	ConsumedTotal:			DINT;				(*$H_R desc := Real time total material consumption for this order; $*)
	ConsumedCart:			DINT;				(*$H_R desc := Real time material consumption from the current cart; $*)
															
END_STRUCT
END_TYPE

// ---- Application/CSP/Customer Interface/csp_customerInterfaces_casePackerCtCall.TcDUT
(*********************************** G.D S.p.A. - Technical Department ***********************************
============= PROGRAM INFO ============
FOLDER:             TBD
MACHINES INVOLVED:  TBD 

============= DESCRIPTION =============
Machine declaration

============= REVISIONS ===============
Date		Version	 	Author      	Description             
----------	-------		------------  	--------------------------------------------
2019/03/27 	0000.00	 	CEC 			Creation of the PRG

**********************************************************************************************************)

TYPE csp_customerInterfaces_casePackerCtCall :
STRUCT
	
	LowCaseSupply:			BOOL;				(*$H_R desc := Connected Technician call - Low Case blank supply; $*)
	LowGlueSupply:			BOOL;				(*$H_R desc := Connected Technician call - Low glue supply; $*)
	LowLabelSupply:			BOOL;				(*$H_R desc := Connected Technician call - Low label supply; $*)
	FullScrapBin:			BOOL;				(*$H_R desc := Connected Technician call - Full machine scrap/waste bin; $*)
	FaultedMain:			BOOL;				(*$H_R desc := Connected Technician call - Main machine is faulted; $*)
	FaultedCaseSupply:		BOOL;				(*$H_R desc := Connected Technician call - Local case blank supply system is faulted; $*)
	TBD1:					BOOL;				(*$H_R desc := Connected Technician call - TBD; $*)
	TBD2:					BOOL;				(*$H_R desc := Connected Technician call - TBD; $*)
	TBD3:					BOOL;				(*$H_R desc := Connected Technician call - TBD; $*)
															
END_STRUCT
END_TYPE

// ---- Application/CSP/Customer Interface/csp_customerInterfaces_casePackerDock.TcDUT
(*********************************** G.D S.p.A. - Technical Department ***********************************
============= PROGRAM INFO ============
FOLDER:             TBD
MACHINES INVOLVED:  TBD 

============= DESCRIPTION =============
Machine declaration

============= REVISIONS ===============
Date		Version	 	Author      	Description             
----------	-------		------------  	--------------------------------------------
2019/03/27 	0000.00	 	CEC 			Creation of the PRG

**********************************************************************************************************)

TYPE csp_customerInterfaces_casePackerDock :
STRUCT
	
	DropAvailable:		BOOL;				(*$H_R desc := Dock [x] is available for cart drop; $*)
	PickAvailable:		BOOL;				(*$H_R desc := Dock [x] is available for cart pick; $*)
	Active:				BOOL;				(*$H_R desc := Dock [x] is actively being consumed; $*)
	EntryReq:			BOOL;				(*$H_RW	act_when := IMMEDIATE ;
														desc := AMR is at Dock [x] and ready to drop or pick; $*)
	EntryAck:			BOOL;				(*$H_R desc := Workcell acknowledge entry request [Future use]; $*)
	EntryOK:			BOOL;				(*$H_R desc := OK for AMR to enter dock; $*)
	AmrExited:			BOOL;				(*$H_RW	act_when := IMMEDIATE ;
														desc := AMR has exited the dock; $*)
															
END_STRUCT
END_TYPE

// ---- Application/CSP/Customer Interface/csp_customerInterfaces_casePackerLabels.TcDUT
(*********************************** G.D S.p.A. - Technical Department ***********************************
============= PROGRAM INFO ============
FOLDER:             TBD
MACHINES INVOLVED:  TBD 

============= DESCRIPTION =============
Machine declaration

============= REVISIONS ===============
Date		Version	 	Author      	Description             
----------	-------		------------  	--------------------------------------------
2019/03/27 	0000.00	 	CEC 			Creation of the PRG

**********************************************************************************************************)

TYPE csp_customerInterfaces_casePackerLabels :
STRUCT
	
	Consumed:						DINT;				(*$H_R desc := Real time total material consumption for this order; $*)
															
END_STRUCT
END_TYPE

// ---- Application/CSP/Customer Interface/csp_customerInterfaces_casePackerProdRej.TcDUT
(*********************************** G.D S.p.A. - Technical Department ***********************************
============= PROGRAM INFO ============
FOLDER:             TBD
MACHINES INVOLVED:  TBD 

============= DESCRIPTION =============
Machine declaration

============= REVISIONS ===============
Date		Version	 	Author      	Description             
----------	-------		------------  	--------------------------------------------
2019/03/27 	0000.00	 	CEC 			Creation of the PRG

**********************************************************************************************************)

TYPE csp_customerInterfaces_casePackerProdRej :
STRUCT
	
	
	Infeed_waterfall:			DINT;				(*$H_R desc := REAL TIME Itemized scrap FOR THIS order; $*)
	Accumulator:				DINT;				(*$H_R desc := REAL TIME Itemized scrap FOR THIS order; $*)
	Case_Feed:					DINT;				(*$H_R desc := REAL TIME Itemized scrap FOR THIS order; $*)
	Discharge:					DINT;				(*$H_R desc := REAL TIME Itemized scrap FOR THIS order; $*)
	TBD5:						DINT;				(*$H_R desc := REAL TIME Itemized scrap FOR THIS order; $*)
	Sample:						DINT;				(*$H_R desc := REAL TIME Itemized scrap FOR THIS order; $*)

															
END_STRUCT
END_TYPE

// ---- Application/CSP/Customer Interface/csp_customerInterfaces_casePackerProduction.TcDUT
(*********************************** G.D S.p.A. - Technical Department ***********************************
============= PROGRAM INFO ============
FOLDER:             TBD
MACHINES INVOLVED:  TBD 

============= DESCRIPTION =============
Machine declaration

============= REVISIONS ===============
Date		Version	 	Author      	Description             
----------	-------		------------  	--------------------------------------------
2019/03/27 	0000.00	 	CEC 			Creation of the PRG

**********************************************************************************************************)

TYPE csp_customerInterfaces_casePackerProduction :
STRUCT
	
	TotalUnits:			DINT;									(*$H_R desc := Real time total number of cartons received for this order; $*)
	GoodPods:			DINT;									(*$H_R desc := Real time total number of good pods packed for this order; $*)
	GoodUnits:			DINT;									(*$H_R desc := Real time total number of good cartons made for this order; $*)
	GoodCases:			DINT;									(*$H_R desc := Real time total number of good cases made for this order; $*)
	TotalUnitsNoReset:	DINT;									(*$H_R desc := Real time total number of cartons received, reset to 1 after 4294967295; $*)
	GoodPodsNoReset:	DINT;									(*$H_R desc := Real time total number of good pods, reset to 1 after 4294967295; $*)
	GoodUnitsNoReset:	DINT;									(*$H_R desc := Real time total number of good cartons, reset to 1 after 4294967295; $*)
	GoodCasesNoReset:	DINT;									(*$H_R desc := Real time total number of good cases, reset to 1 after 4294967295; $*)
	TotalScrapUnits:	DINT;									(*$H_R desc := Real time total number of scrap cartons rejected; $*)
	TotalOrderTime:		DINT;									(*$H_R desc := Real time total minute counter for current order; $*)
	TotalRunningTime:	DINT;									(*$H_R desc := Real time total minute counter for running time in current order; $*)
	PercentScrapUnits:	DINT;									(*$H_R desc := Real time percentage of total cartons rejected; $*)
	Rejects:			csp_customerInterfaces_casePackerProdRej;
															
END_STRUCT
END_TYPE

// ---- Application/CSP/Customer Interface/csp_customerInterfaces_casePackerStart.TcDUT
(*********************************** G.D S.p.A. - Technical Department ***********************************
============= PROGRAM INFO ============
FOLDER:             TBD
MACHINES INVOLVED:  TBD 

============= DESCRIPTION =============
Machine declaration

============= REVISIONS ===============
Date		Version	 	Author      	Description             
----------	-------		------------  	--------------------------------------------
2019/03/27 	0000.00	 	CEC 			Creation of the PRG

**********************************************************************************************************)

TYPE csp_customerInterfaces_casePackerStart :
STRUCT
	
	Request:					BOOL;				(*$H_R desc := Machine request FOR permission TO start; $*)
	Ramp:						BOOL;				(*$H_R desc := Machine is in high current start-up ramp; $*)
	PeakWait:					BOOL;				(*$H_RW	act_when := IMMEDIATE ;
															desc := Request FROM SCADA FOR machine TO delay start; $*)
															
END_STRUCT
END_TYPE

// ---- Application/CSP/Customer Interface/csp_customerInterfaces_casePackerStatus.TcDUT
(*********************************** G.D S.p.A. - Technical Department ***********************************
============= PROGRAM INFO ============
FOLDER:             TBD
MACHINES INVOLVED:  TBD 

============= DESCRIPTION =============
Machine declaration

============= REVISIONS ===============
Date		Version	 	Author      	Description             
----------	-------		------------  	--------------------------------------------
2019/03/27 	0000.00	 	CEC 			Creation of the PRG

**********************************************************************************************************)

TYPE csp_customerInterfaces_casePackerStatus :
STRUCT
	
	Online:					BOOL;				(*$H_R desc := Machine is online; $*)
	Job:					DINT;				(*$H_R desc := Current order (Job) status; $*)
	NextJob:				DINT;				(*$H_R desc := Next order (Job) status; $*)
	Running:				BOOL;				(*$H_R desc := Machine is actively making product; $*)
	Faulted:				csp_customerInterfaces_casePackerStFault;
	RunOut:					BOOL;				(*$H_R desc := Machine AND  conveyor clearance in process; $*)
	RunOutComplete:			BOOL;				(*$H_R desc := Machine AND conveyor clearance complete; $*)
	Rate:					csp_customerInterfaces_casePackerStRate;
	Stop:					csp_customerInterfaces_casePackerStStop;
	Starved:				csp_customerInterfaces_casePackerStStarved;
	Blocked:				csp_customerInterfaces_casePackerStBlocked;
															
END_STRUCT
END_TYPE

// ---- Application/CSP/Customer Interface/csp_customerInterfaces_casePackerStBlocked.TcDUT
(*********************************** G.D S.p.A. - Technical Department ***********************************
============= PROGRAM INFO ============
FOLDER:             TBD
MACHINES INVOLVED:  TBD 

============= DESCRIPTION =============
Machine declaration

============= REVISIONS ===============
Date		Version	 	Author      	Description             
----------	-------		------------  	--------------------------------------------
2019/03/27 	0000.00	 	CEC 			Creation of the PRG

**********************************************************************************************************)

TYPE csp_customerInterfaces_casePackerStBlocked :
STRUCT
	
	Downstream:	BOOL;				(*$H_R desc := Stopped due TO downstream backup; $*)
	Reject:		BOOL;				(*$H_R desc := Stopped due TO scrap backup; $*)
	Waste:		BOOL;				(*$H_R desc := Stopped due TO waste backup; $*)
															
END_STRUCT
END_TYPE

// ---- Application/CSP/Customer Interface/csp_customerInterfaces_casePackerStFault.TcDUT
(*********************************** G.D S.p.A. - Technical Department ***********************************
============= PROGRAM INFO ============
FOLDER:             TBD
MACHINES INVOLVED:  TBD 

============= DESCRIPTION =============
Machine declaration

============= REVISIONS ===============
Date		Version	 	Author      	Description             
----------	-------		------------  	--------------------------------------------
2019/03/27 	0000.00	 	CEC 			Creation of the PRG

**********************************************************************************************************)

TYPE csp_customerInterfaces_casePackerStFault :
STRUCT
	
	Main:				BOOL;				(*$H_R desc := Main machine is faulted; $*)
	CaseBlanks:			BOOL;				(*$H_R desc := Local case blank supply system is faulted; $*)
															
END_STRUCT
END_TYPE

// ---- Application/CSP/Customer Interface/csp_customerInterfaces_casePackerStRate.TcDUT
(*********************************** G.D S.p.A. - Technical Department ***********************************
============= PROGRAM INFO ============
FOLDER:             TBD
MACHINES INVOLVED:  TBD 

============= DESCRIPTION =============
Machine declaration

============= REVISIONS ===============
Date		Version	 	Author      	Description             
----------	-------		------------  	--------------------------------------------
2019/03/27 	0000.00	 	CEC 			Creation of the PRG

**********************************************************************************************************)

TYPE csp_customerInterfaces_casePackerStRate :
STRUCT
	
	Target:			INT;				(*$H_R desc := Target rate in Pods/minute; $*)
	Actual:			INT;				(*$H_R desc := REAL-TIME rate in Pods/minute; $*)
															
END_STRUCT
END_TYPE

// ---- Application/CSP/Customer Interface/csp_customerInterfaces_casePackerStStarved.TcDUT
(*********************************** G.D S.p.A. - Technical Department ***********************************
============= PROGRAM INFO ============
FOLDER:             TBD
MACHINES INVOLVED:  TBD 

============= DESCRIPTION =============
Machine declaration

============= REVISIONS ===============
Date		Version	 	Author      	Description             
----------	-------		------------  	--------------------------------------------
2019/03/27 	0000.00	 	CEC 			Creation of the PRG

**********************************************************************************************************)

TYPE csp_customerInterfaces_casePackerStStarved :
STRUCT
	
	Units:			BOOL;				(*$H_R desc := Carton infeed is empty due to upstream supply; $*)
	CaseBlanks:		BOOL;				(*$H_R desc := Case blank infeed is empty due to upstream supply; $*)
	Glue:			BOOL;				(*$H_R desc := Glue hopper is empty; $*)
	Labels:			BOOL;				(*$H_R desc := Case labeler reel is empty; $*)
															
END_STRUCT
END_TYPE

// ---- Application/CSP/Customer Interface/csp_customerInterfaces_casePackerStStop.TcDUT
(*********************************** G.D S.p.A. - Technical Department ***********************************
============= PROGRAM INFO ============
FOLDER:             TBD
MACHINES INVOLVED:  TBD 

============= DESCRIPTION =============
Machine declaration

============= REVISIONS ===============
Date		Version	 	Author      	Description             
----------	-------		------------  	--------------------------------------------
2019/03/27 	0000.00	 	CEC 			Creation of the PRG

**********************************************************************************************************)

TYPE csp_customerInterfaces_casePackerStStop :
STRUCT
	
	AutoReason:		DINT;				(*$H_R desc := Automatically collected reason FOR current downtime; $*)
	Estop:			BOOL;				(*$H_R desc := Current downtime a result OF Estop; $*)
	Guard:			BOOL;				(*$H_R desc := Current downtime a result OF guard trip; $*)
	Operator:		BOOL;				(*$H_R desc := Current downtime a result OF normal operator stop; $*)
															
END_STRUCT
END_TYPE

// ---- Application/CSP/Customer Interface/csp_customerInterfaces_fillWeight.TcDUT
(*********************************** G.D S.p.A. - Technical Department ***********************************
============= PROGRAM INFO ============
FOLDER:             TBD
MACHINES INVOLVED:  TBD 

============= DESCRIPTION =============
Machine declaration

============= REVISIONS ===============
Date		Version	 	Author      	Description             
----------	-------		------------  	--------------------------------------------
2019/03/27 	0000.00	 	CEC 			Creation of the PRG

**********************************************************************************************************)

TYPE csp_customerInterfaces_fillWeight :
STRUCT
	
	Target:				REAL;				(*$H_RW	act_when := IMMEDIATE ;
															desc := Ingredient fill weight; $*)
	Maximum:			REAL;				(*$H_RW	act_when := IMMEDIATE ;
															desc := Ingredient max weight; $*)
	Minimum:			REAL;				(*$H_RW	act_when := IMMEDIATE ;
															desc := Ingredient min weight; $*)
	
END_STRUCT
END_TYPE

// ---- Application/CSP/Customer Interface/csp_customerInterfaces_mark.TcDUT
(*********************************** G.D S.p.A. - Technical Department ***********************************
============= PROGRAM INFO ============
FOLDER:             TBD
MACHINES INVOLVED:  TBD 

============= DESCRIPTION =============
Machine declaration

============= REVISIONS ===============
Date		Version	 	Author      	Description             
----------	-------		------------  	--------------------------------------------
2019/03/27 	0000.00	 	CEC 			Creation of the PRG

**********************************************************************************************************)

TYPE csp_customerInterfaces_mark :
STRUCT
	
	ID:								STRING;				(*$H_RW	act_when := IMMEDIATE ;
															desc := Print job ID FROM MES; $*)
	BUBD:							csp_customerInterfaces_markBUBD;
		
	OriginDate:						STRING;				(*$H_RW	act_when := IMMEDIATE ;
															desc := DATE the Pod was manufactured; $*)					
	DestCode:						STRING;				(*$H_RW	act_when := IMMEDIATE ;
															desc := Localization code FOR destination; $*)					
	PartnerSite:					STRING;				(*$H_RW	act_when := IMMEDIATE ;
															desc := Partner site code; $*)	
	KdpSite: 						STRING; 			(*$H_RW act_when := IMMEDIATE ;
															desc := KDP site code; $*)				
	Template:						csp_customerInterfaces_markTemplate;
															
															
END_STRUCT
END_TYPE

// ---- Application/CSP/Customer Interface/csp_customerInterfaces_markBUBD.TcDUT
(*********************************** G.D S.p.A. - Technical Department ***********************************
============= PROGRAM INFO ============
FOLDER:             TBD
MACHINES INVOLVED:  TBD 

============= DESCRIPTION =============
Machine declaration

============= REVISIONS ===============
Date		Version	 	Author      	Description             
----------	-------		------------  	--------------------------------------------
2019/03/27 	0000.00	 	CEC 			Creation of the PRG

**********************************************************************************************************)

TYPE csp_customerInterfaces_markBUBD :
STRUCT
	
	BestUsedByDate:			STRING;				(*$H_RW	act_when := IMMEDIATE ;
															desc := Best Used BY DATE; $*)													
	BestUsedByDate_Short:	STRING;				(*$H_RW	act_when := IMMEDIATE ;
															desc := Best Used BY DATE; $*)													
	Prefix:					STRING;				(*$H_RW	act_when := IMMEDIATE ;
															desc := BUBD Prefix (abbreviation); $*)	
	Format:					STRING;				(*$H_RW	act_when := IMMEDIATE ;
															desc := BUBD localized DATE format; $*)		
															
END_STRUCT
END_TYPE

// ---- Application/CSP/Customer Interface/csp_customerInterfaces_markTemplate.TcDUT
(*********************************** G.D S.p.A. - Technical Department ***********************************
============= PROGRAM INFO ============
FOLDER:             TBD
MACHINES INVOLVED:  TBD 

============= DESCRIPTION =============
Machine declaration

============= REVISIONS ===============
Date		Version	 	Author      	Description             
----------	-------		------------  	--------------------------------------------
2019/03/27 	0000.00	 	CEC 			Creation of the PRG

**********************************************************************************************************)

TYPE csp_customerInterfaces_markTemplate :
STRUCT
	
	Pod:					STRING;				(*$H_RW	act_when := IMMEDIATE ;
														desc := Filler product mark template [future use]; $*)				
	Carton:					STRING;				(*$H_RW	act_when := IMMEDIATE ;
														desc := Cartoner product mark template [future use]; $*)					
	CASEPACK:				STRING;				(*$H_RW	act_when := IMMEDIATE ;
														desc := CASE packer product mark template [future use]; $*)	
							
															
END_STRUCT
END_TYPE

// ---- Application/CSP/Customer Interface/csp_customerInterfaces_material.TcDUT
(*********************************** G.D S.p.A. - Technical Department ***********************************
============= PROGRAM INFO ============
FOLDER:             TBD
MACHINES INVOLVED:  TBD 

============= DESCRIPTION =============
Machine declaration

============= REVISIONS ===============
Date		Version	 	Author      	Description             
----------	-------		------------  	--------------------------------------------
2019/03/27 	0000.00	 	CEC 			Creation of the PRG

**********************************************************************************************************)

TYPE csp_customerInterfaces_material :
STRUCT
	
	ID:							STRING;				(*$H_RW	act_when := IMMEDIATE ;
															desc := Material ID in current order; $*)
	QTY:						REAL;				(*$H_RW	act_when := IMMEDIATE ;
															desc := Total expected material QTY for current order; $*)
															
END_STRUCT
END_TYPE

// ---- Application/CSP/Customer Interface/csp_customerInterfaces_MES.TcDUT
(*********************************** G.D S.p.A. - Technical Department ***********************************
============= PROGRAM INFO ============
FOLDER:             TBD
MACHINES INVOLVED:  TBD 

============= DESCRIPTION =============
Machine declaration

============= REVISIONS ===============
Date		Version	 	Author      	Description             
----------	-------		------------  	--------------------------------------------
2019/03/27 	0000.00	 	CEC 			Creation of the PRG

**********************************************************************************************************)

TYPE csp_customerInterfaces_MES :
STRUCT

	StartJobReq:					BOOL;				(*$H_RW	act_when := IMMEDIATE ;
															desc := Request FROM MES TO start the current job; $*)				
	RunOutReq:						BOOL;				(*$H_RW	act_when := IMMEDIATE ;
															desc := Request FROM MES TO execute a line clearance; $*)				
	EndJobReq:						BOOL;				(*$H_RW	act_when := IMMEDIATE ;
															desc := Request FROM MES TO end the current job; $*)					
	CycleEnable:					BOOL;				(*$H_RW	act_when := IMMEDIATE ;
															desc := Premissive FROM MES TO run the line; $*)					
	Alarm:							DINT;				(*$H_RW	act_when := IMMEDIATE ;
															desc := Predefined alarms FROM MES; $*)					
	Warning:						DINT;				(*$H_RW	act_when := IMMEDIATE ;
															desc := Predefined warnings/messages FROM MES; $*)				
															
END_STRUCT
END_TYPE

// ---- Application/CSP/Customer Interface/csp_customerInterfaces_order.TcDUT
(*********************************** G.D S.p.A. - Technical Department ***********************************
============= PROGRAM INFO ============
FOLDER:             TBD
MACHINES INVOLVED:  TBD 

============= DESCRIPTION =============
Machine declaration

============= REVISIONS ===============
Date		Version	 	Author      	Description             
----------	-------		------------  	--------------------------------------------
2019/03/27 	0000.00	 	CEC 			Creation of the PRG

**********************************************************************************************************)

TYPE csp_customerInterfaces_order :
STRUCT
	
	ID:								STRING;				(*$H_RW	act_when := IMMEDIATE ;
															desc := product order identifier; $*)
	SapBatchID:						STRING;				(*$H_RW	act_when := IMMEDIATE ;
															desc := SAP batch ID; $*)
	
END_STRUCT
END_TYPE

// ---- Application/CSP/Customer Interface/csp_customerInterfaces_palletizer.TcDUT
(*********************************** G.D S.p.A. - Technical Department ***********************************
============= PROGRAM INFO ============
FOLDER:             TBD
MACHINES INVOLVED:  TBD 

============= DESCRIPTION =============
Machine declaration

============= REVISIONS ===============
Date		Version	 	Author      	Description             
----------	-------		------------  	--------------------------------------------
2019/03/27 	0000.00	 	CEC 			Creation of the PRG

**********************************************************************************************************)

TYPE csp_customerInterfaces_palletizer :
STRUCT
	
	Ready:				BOOL;			(*$H_RW	act_when := IMMEDIATE ;
															desc := Palletizer is ready to receive cases; $*)
															
END_STRUCT
END_TYPE

// ---- Application/CSP/Customer Interface/csp_customerInterfaces_product.TcDUT
(*********************************** G.D S.p.A. - Technical Department ***********************************
============= PROGRAM INFO ============
FOLDER:             TBD
MACHINES INVOLVED:  TBD 

============= DESCRIPTION =============
Machine declaration

============= REVISIONS ===============
Date		Version	 	Author      	Description             
----------	-------		------------  	--------------------------------------------
2019/03/27 	0000.00	 	CEC 			Creation of the PRG

**********************************************************************************************************)

TYPE csp_customerInterfaces_product :
STRUCT
	
	ID:							STRING;				(*$H_RW	act_when := IMMEDIATE ;
														desc := Product ID; $*)
	UPC:						STRING;				(*$H_RW	act_when := IMMEDIATE ;
														desc := Product UPC; $*)
	
	PodsPerCarton: 				INT;				(*$H_RW	act_when := IMMEDIATE ;
															desc := recipe data, number of cups inside a carton; $*)
	
	PodsPerCase:				INT;				(*$H_RW	act_when := IMMEDIATE ;
															desc := recipe data, number of cups inside a case; $*)
	CartonsPerCase:				INT;				(*$H_RW	act_when := IMMEDIATE ;
															desc := recipe data, number of cartons inside a case; $*)

	FillWeight:					csp_customerInterfaces_fillWeight;

	FilterType:					STRING;				(*$H_RW	act_when := IMMEDIATE ;
															desc := Filter type; $*)
	CaffeinatedFlag:			BOOL;				(*$H_RW	act_when := IMMEDIATE ;
															desc := Coffee Caffeinated flag; $*)
	KosherFlag:					BOOL;				(*$H_RW	act_when := IMMEDIATE ;
															desc := Coffee Kosher flag; $*)
	OrganicFlag:				BOOL;				(*$H_RW	act_when := IMMEDIATE ;
															desc := Coffee Organic flag; $*)
	FlavorFlag:					BOOL;				(*$H_RW	act_when := IMMEDIATE ;
															desc := Coffee Flavored flag; $*)
	FlavorDose:					REAL;				(*$H_RW	act_when := IMMEDIATE ;
															desc := Coffee inline flavor dose [future use]; $*)
	ShelfLife:					INT;				(*$H_RW	act_when := IMMEDIATE ;
															desc := Pod shelf life; $*)
	
END_STRUCT
END_TYPE

// ---- Application/CSP/Customer Interface/csp_customerInterfaces_recipe.TcDUT
(*********************************** G.D S.p.A. - Technical Department ***********************************
============= PROGRAM INFO ============
FOLDER:             TBD
MACHINES INVOLVED:  TBD 

============= DESCRIPTION =============
Machine declaration

============= REVISIONS ===============
Date		Version	 	Author      	Description             
----------	-------		------------  	--------------------------------------------
2019/03/27 	0000.00	 	CEC 			Creation of the PRG

**********************************************************************************************************)

TYPE csp_customerInterfaces_recipe :
STRUCT
	
	Filler:								STRING;				(*$H_RW	act_when := IMMEDIATE ;
															desc := Filler recipe ID [future use]; $*)
	Cartoner:							STRING;				(*$H_RW	act_when := IMMEDIATE ;
															desc := Cartoner recipe ID [future use]; $*)
	CasePacker:							STRING;				(*$H_RW	act_when := IMMEDIATE ;
															desc := Case packer recipe ID [future use]; $*)
															
END_STRUCT
END_TYPE

// ---- Application/CSP/Main/AccU Change/csp_main_accuChange_constant.TcDUT
TYPE csp_main_accuChange_constant :
STRUCT
	(*BELT Info*)
	MIN_VELOCITY_MMpSEC:						LREAL := 100;
	MAX_VELOCITY_MMpSEC:						LREAL := 666.5487;
	MAX_ACCELERATION_MMpSEC2:					LREAL := 1000;
	MAX_DECELERATION_MMpSEC2:					LREAL := 1000;
	MAX_JERK_MMpSEC3:							LREAL := 100000;
	RUNNING_ACCELERATION_MMMpSEC2:				LREAL := 3000;
	RUNNING_DECELERATION_MMpSEC2:				LREAL := 3000;
	MAX_FOLLOWING_ERROR_MM:						LREAL := 5;
	
	RUNNING_JERK_MMpSEC3:						LREAL := 1000000;
	MOTOR_MAX_VELOCITY_DEGPS:					LREAL := 9600;
	MOTOR_MAX_ACCELERATION_DEGPS2:				LREAL := 4800;
	MOTOR_MAX_DECELERATION_DEGPS2:				LREAL := 4800;
	MOTOR_MAX_JERK_DEGPS3:						LREAL := 100000000; 
	MOTOR_MAX_FOLLOWING_ERROR_DEG:				LREAL := 2;
END_STRUCT
END_TYPE

// ---- Application/CSP/Main/AccU Change/csp_main_accuChange_enum.TcDUT
TYPE csp_main_accuChange_enum :
(
	CSP_MAIN_ACCUCHANGE_STATUS_BRAND_CHECK 									:= 0,
	CSP_MAIN_ACCUCHANGE_STATUS_BRAND_CHANGE_REQUEST 						:= 5,
	CSP_MAIN_ACCUCHANGE_STATUS_PRODUCT_REMOVED_CHECK 						:= 10,
	CSP_MAIN_ACCUCHANGE_STATUS_RESET_REQUEST								:= 20,
	CSP_MAIN_ACCUCHANGE_STATUS_SAFE_POSITION_REQUEST 						:= 30,
	CSP_MAIN_ACCUCHANGE_STATUS_OPERATOR_REPLACE_CHANGE_PARTS 				:= 40,
	CSP_MAIN_ACCUCHANGE_STATUS_CHANGE_PARTS_REPLACED						:= 50,
	CSP_MAIN_ACCUCHANGE_STATUS_VERIFYING_CHANGE_PARTS_START					:= 60,
	CSP_MAIN_ACCUCHANGE_STATUS_VERIFYING_CASE_FEED_EOAT						:= 61,
	CSP_MAIN_ACCUCHANGE_STATUS_VERIFYING_LOADER_PUSHER						:= 62,
	CSP_MAIN_ACCUCHANGE_STATUS_VERIFYING_LOADER_GUIDE_PLATE					:= 63,
	CSP_MAIN_ACCUCHANGE_STATUS_VERIFYING_CLOSING_PADDLES					:= 64,
	CSP_MAIN_ACCUCHANGE_STATUS_VERIFYING_ALL_RFID							:= 65,
	CSP_MAIN_ACCUCHANGE_STATUS_GROUP_1_ACCU_MOVE_REQUEST 					:= 70,
	CSP_MAIN_ACCUCHANGE_STATUS_GROUP_2_TR_UP_ACCU_MOVE_REQUEST 				:= 80,
	CSP_MAIN_ACCUCHANGE_STATUS_GROUP_2_TR_DOWN_ACCU_MOVE_REQUEST 			:= 85,
	CSP_MAIN_ACCUCHANGE_STATUS_ADD_CASE_BLANKS 								:= 100,
	CSP_MAIN_ACCUCHANGE_STATUS_DONE											:= 900
) := CSP_MAIN_ACCUCHANGE_STATUS_BRAND_CHECK;
END_TYPE

// ---- Application/CSP/Main/AccU Change/csp_main_accuChange_partColor_enum.TcDUT
TYPE csp_main_accuChange_partColor_enum :
(
	NO_COLOR		 	:= 0,
	RED					:= 1,
	GREEN				:= 2,
	BLUE				:= 3,
	YELLOW				:= 4,
	WHITE				:= 5,
	BLACK				:= 6,
	ORANGE				:= 7
);
END_TYPE

// ---- Application/CSP/Main/AccU Change/csp_main_accuChange_RFID_reader_list.TcDUT
TYPE csp_main_accuChange_RFID_reader_list :
(
	NO_READER_SELECTED							:= 0,
	CASE_FEED_EOAT_READER						:= 1,
	LOADER_PUSHER_READER						:= 2, (* IN CODE *)
	LOADER_GUIDE_PLATE_READER					:= 3, (* IN CODE *)
	CLOSING_PADDLES_READER						:= 4  (* IN CODE *)
):= NO_READER_SELECTED;
END_TYPE

// ---- Application/CSP/Main/AccU Change/csp_main_accuChange_RFID_read_write_status.TcDUT
TYPE csp_main_accuChange_RFID_read_write_status :
(
	READ_WRITE_STATUS_START_RFID_READ						:= 0,
	READ_WRITE_STATUS_SEND_READ_COMMAND						:= 1,
	READ_WRITE_STATUS_WAIT_FOR_READ_RESULT					:= 2,
	READ_WRITE_STATUS_CHECK_READ_RESULT						:= 3,
	
	READ_WRITE_STATUS_START_RFID_WRITE						:= 101,
	READ_WRITE_STATUS_SEND_WRITE_COMMAND					:= 102,
	READ_WRITE_STATUS_WAIT_FOR_WRITE_SUCCESS				:= 103,
	READ_WRITE_STATUS_WRITE_TO_READ							:= 104,
	
	READ_WRITE_STATUS_WAITING								:= 900,
	READ_WRITE_STATUS_ERROR									:= 999
):= READ_WRITE_STATUS_WAITING;
END_TYPE

// ---- Application/CSP/Main/AccU Change/csp_main_accuChange_RFID_running_check_status.TcDUT
TYPE csp_main_accuChange_RFID_running_check_status :
(
	READ_RUNNING_CHECK_STATUS_START									:= 0,
	READ_RUNNING_CHECK_STATUS_EOAT_CHECK_CP							:= 1,
	READ_RUNNING_CHECK_STATUS_EOAT_SEND_READ						:= 2,
	READ_RUNNING_CHECK_STATUS_EOAT_CHECK_READ						:= 3,
	READ_RUNNING_CHECK_STATUS_LOADER_PUSHER_CHECK_CP				:= 4,
	READ_RUNNING_CHECK_STATUS_LOADER_PUSHER_SEND_READ				:= 5,
	READ_RUNNING_CHECK_STATUS_LOADER_PUSHER_CHECK_READ				:= 6,
	READ_RUNNING_CHECK_STATUS_LOADER_PLATE_CHECK_CP					:= 7,
	READ_RUNNING_CHECK_STATUS_LOADER_PLATE_SEND_READ				:= 8,
	READ_RUNNING_CHECK_STATUS_LOADER_PLATE_CHECK_READ				:= 9,
	
	READ_RUNNING_CHECK_STATUS_DONE									:= 900,
	READ_RUNNING_CHECK_STATUS_WAITING								:= 950,
	READ_RUNNING_CHECK_STATUS_ERROR									:= 999
):= READ_RUNNING_CHECK_STATUS_WAITING;
END_TYPE

// ---- Application/CSP/Main/Brand/csp_main_brand_cam_change.TcDUT
TYPE csp_main_brand_cam_change :
(
	CSP_MAIN_BRAND_CAM_CHANGE_INIT 							:= 0,
	CSP_MAIN_BRAND_CAM_CHANGE_PHASE_LOAD 					:= 10,
	CSP_MAIN_BRAND_CAM_CHANGE_PHASE_TRANSFER 				:= 20,
	CSP_MAIN_BRAND_CAM_CHANGE_CONNEECTION_LOAD 				:= 30,
	CSP_MAIN_BRAND_CAM_CHANGE_CONNECTION_TRANSFER 			:= 40,		
	CSP_MAIN_BRAND_CAM_CHANGE_DONE							:= 900,
	CSP_MAIN_BRAND_CAM_CHANGE_ERROR							:= 999
) := CSP_MAIN_BRAND_CAM_CHANGE_INIT;
END_TYPE

// ---- Application/CSP/Main/Brand/csp_main_brand_carton_format_enum.TcDUT
TYPE csp_main_brand_carton_format_enum :
	(
		csp_MAIN_BRAND_X_COUNT_XxXCARTON_X_COUNT_CASE  	:= 0,
		csp_MAIN_BRAND_6_COUNT_2x3CARTON_6_COUNT_CASE  	:= 1,
		csp_MAIN_BRAND_8_COUNT_2x4CARTON_6_COUNT_CASE  	:= 2,
		csp_MAIN_BRAND_10_COUNT_2x3CARTON_6_COUNT_CASE	:= 3,
		csp_MAIN_BRAND_12_COUNT_2x3CARTON_6_COUNT_CASE	:= 4,
		csp_MAIN_BRAND_16_COUNT_2x3CARTON_4_COUNT_CASE	:= 5,
		csp_MAIN_BRAND_18_COUNT_2x3CARTON_4_COUNT_CASE	:= 6,
		csp_MAIN_BRAND_14_COUNT_2x4CARTON_6_COUNT_CASE	:= 7,
		csp_MAIN_BRAND_16_COUNT_2x4CARTON_6_COUNT_CASE	:= 8,
		csp_MAIN_BRAND_20_COUNT_2x4CARTON_4_COUNT_CASE	:= 9,
		csp_MAIN_BRAND_22_COUNT_2x4CARTON_4_COUNT_CASE	:= 10,
		csp_MAIN_BRAND_24_COUNT_2x4CARTON_4_COUNT_CASE	:= 11,
		csp_MAIN_BRAND_28_COUNT_2x4CARTON_4_COUNT_CASE	:= 12,
		csp_MAIN_BRAND_30_COUNT_2x4CARTON_4_COUNT_CASE	:= 13,
		csp_MAIN_BRAND_32_COUNT_2x4CARTON_4_COUNT_CASE	:= 14,
		csp_MAIN_BRAND_34_COUNT_3x4CARTON_4_COUNT_CASE	:= 15,
		csp_MAIN_BRAND_36_COUNT_3x4CARTON_4_COUNT_CASE	:= 16,		
		csp_MAIN_BRAND_44_COUNT_3x4CARTON_4_COUNT_CASE	:= 17,
		csp_MAIN_BRAND_46_COUNT_3x4CARTON_4_COUNT_CASE	:= 18,
		csp_MAIN_BRAND_48_COUNT_3x4CARTON_4_COUNT_CASE	:= 19
	
	) := csp_MAIN_BRAND_X_COUNT_XxXCARTON_X_COUNT_CASE;
END_TYPE

// ---- Application/CSP/Main/Brand/csp_main_brand_case_pattern.TcDUT
TYPE csp_main_brand_case_pattern :
STRUCT
	
	case_pattern_L:								INT := 2; (*$P min := 0; max := 5; step := 1; unit := u ; desc := Case Pattern L; $*)
	case_pattern_W:								INT := 2; (*$P min := 0; max := 5; step := 1; unit := u; desc := Case Pattern W; $*)
	case_pattern_D:								INT := 1; (*$P min := 0; max := 5; step := 1; unit := u; desc := Case Pattern D; $*)
			
END_STRUCT
END_TYPE

// ---- Application/CSP/Main/Brand/csp_main_brand_product_dimension.TcDUT
TYPE csp_main_brand_product_dimension :
	STRUCT
		
		carton_size_L_mm:								LREAL := 100; (*$P min := 0; max := 200; step := 0.1; unit :=  mm; desc := Carton Length; $*)
		carton_size_W_mm:								LREAL := 100; (*$P min := 0; max := 200; step := 0.1; unit :=  mm; desc := Carton Width; $*)
		carton_size_D_mm:								LREAL := 100; (*$P min := 0; max := 200; step := 0.1; unit :=  mm; desc := Carton Depth; $*)
				
	END_STRUCT
END_TYPE

// ---- Application/CSP/Main/Interface/csp_main_interface_csv_read.TcDUT
{attribute 'qualified_only'}
{attribute 'strict'}
TYPE csp_main_interface_csv_read :
(
	
	csv_read_idle					:= 0,
	csv_read_wait_for_alarm			:= 10,
	csv_read_clear_variables		:= 20,
	csv_read_trim_object_name		:= 30,
	csv_read_open_csv_file			:= 40,
	csv_read_verify_open			:= 50,
	csv_read_read_csv_file			:= 60,
	csv_read_verify_read			:= 70,
	csv_read_parse_csv_stop_data	:= 80,
	csv_read_compare_stop			:= 90,
	csv_read_alarm_found			:= 100,
	csv_read_close_csv_file			:= 200,
	csv_read_close_csv_file_verify	:= 210
	
) := csv_read_idle;
END_TYPE

// ---- Application/CSP/Main/Jog Manager/csp_jog_accu_suggested_speeds.TcDUT
TYPE csp_jog_accu_suggested_speeds :
	STRUCT
		NO_UAXIS_SELECT_TO_JOG_SPEED:															LREAL := 0;
		SMTR61700_TRANSFER_INFEED_DEPTH_SPEED:													LREAL := 1.5;
		SMTR61710_TRANSFER_INFEED_WATERFALL_ADJUST_SPEED:										LREAL := 1;
		SMTR61720_SMTR61730_TRANSFER_ACCUMULATOR_DEPTH_AND_CONVEYOR_DEPTH_SPEED:				LREAL := 1;
		SMTR61510_CASE_TOP_RAIL_DEPTH_SPEED:													LREAL := 2;
		SMTR61430_SMTR61500_CASE_TOP_RAIL_LS_AND_OS_WIDTH_SPEED:								LREAL := 1;
		SMTR61210_SMTR61200_SMTR61420_CASE_FEED_SHUTTLE_TRANSPORT_AND_DISCHARGE_DEPTH_SPEED:	LREAL := 2;
		SMTR61220_CASE_FEED_MAGAZINE_LS_DEPTH_SPEED:											LREAL := 1;
		SMTR61230_CASE_FEED_MAGAZINE_OS_DEPTH_SPEED:											LREAL := 1;
		SMTR61300_CASE_LOADER_GUIDE_WIDTH_SPEED:												LREAL := 5;
		SMTR61410_CASE_GLUE_LS_LOWER_POSITION_SPEED:											LREAL := 3;
		SMTR61400_CASE_GLUE_LS_UPPER_POSITION_SPEED:											LREAL := 3;
		SMTR61330_CASE_GLUE_OS_LOWER_POSITION_SPEED:											LREAL := 3;
		SMTR61320_CASE_GLUE_OS_UPPER_POSITION_SPEED:											LREAL := 3;
		SMTR61310_CASE_GLUE_OS_WIDTH_SPEED:														LREAL := 3;
		
		(*Tie AccuChange axis list enum to each axis' suggested speed
		If accuchange jog list enum is changed, indices here must be adjusted accordingly*)
		Suggested_Speeds:	ARRAY[JOG_MANAGER_JOG_LIST_NONE..JOG_MANAGER_JOG_LIST_MAX] OF LREAL :=
			[NO_UAXIS_SELECT_TO_JOG_SPEED, //0
			SMTR61700_TRANSFER_INFEED_DEPTH_SPEED, //1
			SMTR61710_TRANSFER_INFEED_WATERFALL_ADJUST_SPEED, //2
			SMTR61720_SMTR61730_TRANSFER_ACCUMULATOR_DEPTH_AND_CONVEYOR_DEPTH_SPEED, //3
			0, //4 - csp_jog_list_AccUChange enum has no 4 value
			SMTR61510_CASE_TOP_RAIL_DEPTH_SPEED, //5
			SMTR61430_SMTR61500_CASE_TOP_RAIL_LS_AND_OS_WIDTH_SPEED, //6
			SMTR61210_SMTR61200_SMTR61420_CASE_FEED_SHUTTLE_TRANSPORT_AND_DISCHARGE_DEPTH_SPEED, //7
			SMTR61220_CASE_FEED_MAGAZINE_LS_DEPTH_SPEED, //8
			SMTR61230_CASE_FEED_MAGAZINE_OS_DEPTH_SPEED, //9
			SMTR61300_CASE_LOADER_GUIDE_WIDTH_SPEED, //10
			SMTR61410_CASE_GLUE_LS_LOWER_POSITION_SPEED, //11
			SMTR61400_CASE_GLUE_LS_UPPER_POSITION_SPEED, //12
			SMTR61330_CASE_GLUE_OS_LOWER_POSITION_SPEED, //13
			SMTR61320_CASE_GLUE_OS_UPPER_POSITION_SPEED, //14
			SMTR61310_CASE_GLUE_OS_WIDTH_SPEED]; //15
	
	END_STRUCT
END_TYPE

// ---- Application/CSP/Main/Jog Manager/csp_jog_list_AccUChange.TcDUT
TYPE csp_jog_list_AccUChange :
(	
	JOG_LIST_NO_UAXIS_SELECT_TO_JOG													:= 0,
	SMTR61700_TRANSFER_INFEED_DEPTH													:= 1,
	SMTR61710_TRANSFER_INFEED_WATERFALL_ADJUST										:= 2,
	SMTR61720_SMTR61730_TRANSFER_ACCUMULATOR_DEPTH_AND_CONVEYOR_DEPTH 				:= 3,
	SMTR61510_CASE_TOP_RAIL_DEPTH													:= 5,
	SMTR61430_SMTR61500_CASE_TOP_RAIL_LS_AND_OS_WIDTH								:= 6,
	SMTR61210_SMTR61200_SMTR61420_CASE_FEED_SHUTTLE_TRANSPORT_AND_DISCHARGE_DEPTH	:= 7,
	SMTR61220_CASE_FEED_MAGAZINE_LS_DEPTH											:= 8,
	SMTR61230_CASE_FEED_MAGAZINE_OS_DEPTH											:= 9,
	SMTR61300_CASE_LOADER_GUIDE_WIDTH												:= 10,
	SMTR61410_CASE_GLUE_LS_LOWER_POSITION											:= 11,
	SMTR61400_CASE_GLUE_LS_UPPER_POSITION											:= 12,
	SMTR61330_CASE_GLUE_OS_LOWER_POSITION											:= 13,
	SMTR61320_CASE_GLUE_OS_UPPER_POSITION											:= 14,
	SMTR61310_CASE_GLUE_OS_WIDTH													:= 15
) := JOG_LIST_NO_UAXIS_SELECT_TO_JOG;
END_TYPE

// ---- Application/CSP/Main/Jog Manager/csp_jog_list_real.TcDUT
TYPE csp_jog_list_real :
(	
	JOG_LIST_NO_RAXIS_SELECT_TO_JOG					:= 0,
	SMTR41323_TRANSFER_ACCUMULATOR_BELT				:= 1, 
	SMTR41223_TRANSFER_ACCUMULATOR_FINGER_LS		:= 2,
	SMTR41203_TRANSFER_ACCUMULATOR_FINGER_OS		:= 3,
	SMTR41103_TRANSFER_ACCUMULATOR_LIFT				:= 4,
	SMTR41503_TRANSFER_CROSSPUSHER_FOLLOWER			:= 10, 
	SMTR41423_TRANSFER_CROSSPUSHER_HORIZONTAL		:= 11,
	SMTR41523_TRANSFER_CROSSPUSHER_VERTICAL			:= 12,	
	SMTR41403_TRANSFER_UPSTACKER_DOWNSTREAM			:= 20,
	SMTR41303_TRANSFER_UPSTACKER_UPSTREAM			:= 21,
	SMTR2103_CASE_TRANSPORT_OS_LEADING				:= 22,
	SMTR2123_CASE_TRANSPORT_OS_TRAILING				:= 23,
    SMTR2203_CASE_TRANSPORT_LS_LEADING				:= 24,
	SMTR2223_CASE_TRANSPORT_LS_TRAILING				:= 25,
    SMTR26103_CASE_TOP_RAIL_SQUARING_LS_TRAILING	:= 26,
	SMTR26123_CASE_TOP_RAIL_SQUARING_LS_LEADING		:= 27,
    SMTR26003_CASE_TOP_RAIL_SQUARING_OS_TRAILING	:= 28,
	SMTR26023_CASE_TOP_RAIL_SQUARING_OS_LEADING		:= 29,
    SMTR2403_CASE_CLOSING_OS_HORIZONTAL				:= 30,
    SMTR2303_CASE_CLOSING_OS_UPPER					:= 31,
    SMTR2323_CASE_CLOSING_OS_LOWER					:= 32,
    SMTR2523_CASE_CLOSING_LS_HORIZONTAL				:= 33,
    SMTR2423_CASE_CLOSING_LS_UPPER					:= 34,
    SMTR2503_CASE_CLOSING_LS_LOWER					:= 35,
    SMTR10423_CASE_FC_LS_LOWER_FOLLWER				:= 36,
    SMTR10403_CASE_FC_LS_LOWER_SPREADER				:= 37,
    SMTR8123_CASE_FC_LS_LOWER_TRAILING_CLOSER   	:= 38,
	SMTR10303_CASE_FC_LS_UPPER_FOLLWER				:= 39,
    SMTR10323_CASE_FC_LS_UPPER_LEADING_MINOR_CLOSER := 40,
	SMTR10223_CASE_FC_LS_UPPER_SPREADER				:= 42,
	SMTR10123_CASE_FC_OS_LOWER_FOLLWER				:= 43,
    SMTR10103_CASE_FC_OS_LOWER_SPREADER				:= 44,
   	SMTR10023_CASE_FC_OS_UPPER_FOLLWER				:= 46,
    SMTR10003_CASE_FC_OS_UPPER_SPREADER				:= 48,
    SMTR8003_CASE_FEED_SHUTTLE_HORIZONTAL			:= 49,
	SMTR8023_CASE_FEED_SHUTTLE_VERTICAL 			:= 50,
    SMTR8323_CASE_LOADER_GUIDE_DOWNSTREAM			:= 51,
    SMTR8523_CASE_LOADER_GUIDE_LENGTH				:= 52,
    SMTR8223_CASE_LOEADER_GUIDE_UPSTREAM	  		:= 53,
    SMTR8503_CASE_LOADER_PUSHER						:= 54,
	SMTR12023_CASE_DISCHARGE_LS_SPEEDBELT			:= 55, 
	SMTR12003_CASE_DISCHARGE_OS_SPEEDBELT			:= 56
	
) := JOG_LIST_NO_RAXIS_SELECT_TO_JOG;
END_TYPE

// ---- Application/CSP/Main/Jog Manager/csp_jog_list_virtual.TcDUT
TYPE csp_jog_list_virtual :
(	
	JOG_LIST_NO_VAXIS_SELECT_TO_JOG				:= 0,
	JOG_LIST_TRANSFER_VIRTUAL					:= 2, 
	JOG_LIST_TRANSFER_ACCUMULATOR_VIRTUAL		:= 12, 
	JOG_LIST_TRANSFER_CROSSPUSHER_VIRTUAL		:= 13,
	JOG_LIST_TRANSFER_UPSTACKER_VITUAL			:= 22,
	JOG_LIST_CSP_CASE_FEED_VIRTUAL				:= 31,
	JOG_LIST_CSP_CASE_TRANSPORT_VIRTUAL			:= 32,
	JOG_LIST_CSP_CASE_LOADER_VIRTUAL			:= 33,
	JOG_LIST_CSP_CASE_VIRTUAL					:= 34	
	
) := JOG_LIST_NO_VAXIS_SELECT_TO_JOG;
END_TYPE

// ---- Application/CSP/Main/Motorization/Snapshot/csp_main_motorization_snapshot.TcDUT
(*********************************** G.D S.p.A. - Technical Department ***********************************
============= PROGRAM INFO ============
FOLDER:             TBD
MACHINES INVOLVED:  TBD 

============= DESCRIPTION =============
csp main motorization manager snapshot struct definition

============= REVISIONS ===============
Date		Version	 	Author      	Description             
----------	-------		------------  	--------------------------------------------
2019/04/27 	0000.00	 	M.Grasso		Creation of the PRG

**********************************************************************************************************)

(*$S desc := Snapshot; $*)
TYPE 
	csp_main_motorization_snapshot:	STRUCT
		message:            message;
		reason:             STRING := '';			(*$ It contains detailed information abaout axis faults $*)
		connection_status:	INT;					(*$ It contains information about the connection status when the message is switched on $*)
END_STRUCT
END_TYPE

// ---- Application/CSP/Main/Motorization/csp_main_motorization_connection_status_enum.TcDUT
(*********************************** G.D S.p.A. - Technical Department ***********************************
============= PROGRAM INFO ============
FOLDER:             TBD
MACHINES INVOLVED:  TBD 

============= DESCRIPTION =============
csp main motorization connection status enum data structure definition

============= REVISIONS ===============
Date		Version	 	Author      	Description             
----------	-------		------------  	--------------------------------------------
2019/04/27 	0000.00	 	M.Grasso		Creation of the PRG

**********************************************************************************************************)

TYPE csp_main_motorization_connection_status_enum :
(
	csp_MAIN_MOTORIZATION_CONNECTION_STATUS_ENUM_IDLE_STATUS_0											:= 0,
	csp_MAIN_MOTORIZATION_CONNECTION_STATUS_ENUM_AXIS_DISABLE_STATUS_10									:= 10,
	csp_MAIN_MOTORIZATION_CONNECTION_STATUS_ENUM_VIRTUAL_MANAGER_REDEFINE_POS_REQ_STATUS_20				:= 20,
	csp_MAIN_MOTORIZATION_CONNECTION_STATUS_ENUM_VIRTUAL_MANAGER_POS_REDEFINING_STATUS_30				:= 30,	
	csp_MAIN_MOTORIZATION_CONNECTION_STATUS_ENUM_VIRTUAL_AXIS_ENABLE_STATUS_40							:= 40,
	csp_MAIN_MOTORIZATION_CONNECTION_STATUS_ENUM_CONNECTION_DONE_STATUS_900								:= 900,
	csp_MAIN_MOTORIZATION_CONNECTION_STATUS_ENUM_CONNECTION_NOT_COMPLETED_STATUS_999					:= 999		
)	:= csp_MAIN_MOTORIZATION_CONNECTION_STATUS_ENUM_CONNECTION_NOT_COMPLETED_STATUS_999;
END_TYPE

// ---- Application/CSP/csp_sw_configurator_struct.TcDUT
(*********************************** G.D S.p.A. - Technical Department ***********************************
============= PROGRAM INFO ============


============= DESCRIPTION =============


============= REVISIONS ===============
Date		Version	 	Author      	Description             
----------	-------		------------  	--------------------------------------------
2019/04/24 	0000.00	 	CEC 			Creation of the PRG

**********************************************************************************************************)

TYPE csp_sw_configurator_struct :
STRUCT


(****************************************************************************************************************************************************)
(*	 COMMON CONFIGURATIONS																																*)
(****************************************************************************************************************************************************)

(****************************************************************************************************************************************************)
(*	 GROUPS CONFIGURATION STRUCT																													*)
(****************************************************************************************************************************************************)
	csp_INTERFACE:												csp_main_configurator_struct;

(****************************************************************************************************************************************************)
(*	 MACHINE OPTIONS																																*)
(****************************************************************************************************************************************************)

	INTERNAL_TESTING:											BOOL := FALSE;	(* BYPASS *)
END_STRUCT
END_TYPE

// ---- Application/CSP/Main/csp_main_configurator_struct.TcDUT
(*********************************** G.D S.p.A. - Technical Department ***********************************
============= PROGRAM INFO ============
FOLDER:             TBD
MACHINES INVOLVED:  TBD 

============= DESCRIPTION =============
csp machine configurator data structure declaration

============= REVISIONS ===============
Date		Version	 	Author      	Description             
----------	-------		------------  	--------------------------------------------
2019/04/24 	0000.00	 	M.Grasso		Creation of the PRG

**********************************************************************************************************)

TYPE csp_main_configurator_struct:
STRUCT
	motman_ref:																POINTER TO motorization_manager;
	machine_ref:															POINTER TO machine;
	service_stop_reclassification_present:									BOOL := TRUE;
END_STRUCT
END_TYPE

// ---- Application/CSP/Main/Phase Manager/csp_main_phaseManager_status_enum.TcDUT
(*********************************** G.D S.p.A. - Technical Department ***********************************
============= PROGRAM INFO ============
FOLDER:             TBD
MACHINES INVOLVED:  TBD 

============= DESCRIPTION =============
WN main phase manager status enum data structure definition

============= REVISIONS ===============
Date		Version	 	Author      	Description             
----------	-------		------------  	--------------------------------------------
2020/06/16 	0000.00	 	G.Cera 			Creation of the PRG

**********************************************************************************************************)

TYPE csp_main_phaseManager_status_enum :
(
	CSP_MAIN_PHASE_MANAGER_STATUS_UNDEFINED_0							:= 0,
	CSP_MAIN_PHASE_MANAGER_STATUS_START_JOB_10							:= 10,
	CSP_MAIN_PHASE_MANAGER_STATUS_STEADY_STATE_20						:= 20,
	CSP_MAIN_PHASE_MANAGER_MANUAL_STEADY_STATE_40						:= 40,
	CSP_MAIN_PHASE_MANAGER_STATUS_NEAR_END_OF_RUN_50					:= 50,
	CSP_MAIN_PHASE_MANAGER_STATUS_RUNOUT_60								:= 60,
	CSP_MAIN_PHASE_MANAGER_STATUS_END_JOB_70							:= 70
) := CSP_MAIN_PHASE_MANAGER_STATUS_UNDEFINED_0;
END_TYPE

// ---- Application/CSP/Main/Phase Manager/Snapshot/csp_main_phaseManager_snapshot.TcDUT
(*********************************** G.D S.p.A. - Technical Department ***********************************
============= PROGRAM INFO ============
FOLDER:             TBD
MACHINES INVOLVED:  TBD 

============= DESCRIPTION =============
WU phase manager snapshot struct definition

============= REVISIONS ===============
Date		Version	 	Author      	Description             
----------	-------		------------  	--------------------------------------------
2020/06/19 	0000.00	 	G.Cera 			Creation of the PRG

**********************************************************************************************************)

(*$S desc := Snapshot; $*)
TYPE 
	csp_main_phaseManager_snapshot:	STRUCT
		message:            	message;
		reason:             	STRING := '';			(*$ It contains detailed information abaout faults $*)
		job_not_scheduled:		BOOL;
		job_pending:			BOOL;
END_STRUCT
END_TYPE

// ---- Application/CSP/Main/Phase Manager/Snapshot/csp_main_phaseManager_warning_snapshot.TcDUT
(*********************************** G.D S.p.A. - Technical Department ***********************************
============= PROGRAM INFO ============
FOLDER:             TBD
MACHINES INVOLVED:  TBD 

============= DESCRIPTION =============
WU phase manager snapshot struct definition

============= REVISIONS ===============
Date		Version	 	Author      	Description             
----------	-------		------------  	--------------------------------------------
2020/06/19 	0000.00	 	G.Cera 			Creation of the PRG

**********************************************************************************************************)

(*$S desc := Snapshot; $*)
TYPE 
	csp_main_phaseManager_warning_snapshot:	STRUCT
		message:            	message;
		w_reason:             	STRING := '';			(*$ It contains detailed information abaout faults $*)
		maintenance_job_active:	BOOL;
END_STRUCT
END_TYPE

// ---- Application/CSP/Main/Phase Manager/Snapshot/csp_main_phMan_start_job_snapshot.TcDUT
(*********************************** G.D S.p.A. - Technical Department ***********************************
============= PROGRAM INFO ============
FOLDER:             TBD
MACHINES INVOLVED:  TBD 

============= DESCRIPTION =============
WU phase manager snapshot struct definition

============= REVISIONS ===============
Date		Version	 	Author      	Description             
----------	-------		------------  	--------------------------------------------
2020/06/19 	0000.00	 	G.Cera 			Creation of the PRG

**********************************************************************************************************)

(*$S desc := Snapshot; $*)
TYPE 
	csp_main_phMan_start_job_snapshot:	STRUCT
		message:            	message;
		sj_reason:             	STRING := '';			(*$ It contains detailed information abaout axis faults $*)
		order_valid:			BOOL;
		product_valid:			BOOL;
		recipe_valid:			BOOL;
		materials_valid:		BOOL;
		mark_valid:				BOOL;
END_STRUCT
END_TYPE

// ---- Application/CSP/Main/Services/RFID FB/ST_BIS00LH_Inputs.TcDUT
TYPE ST_BIS00LH_Inputs :
STRUCT
	DeviceDiag AT %I*: BOOL;
	DeviceState AT %I*: BOOL;
	ChannelState AT %I*: USINT;
	InfoDataState AT %I*: UINT;
	ByteArr AT %I*: ARRAY[0..9] OF BYTE;
END_STRUCT
END_TYPE

// ---- Application/CSP/Main/Services/RFID FB/ST_BIS00LH_IO.TcDUT
TYPE ST_BIS00LH_IO :
STRUCT
	IN: ST_BIS00LH_Inputs;
	OUT: ST_BIS00LH_Outputs;
END_STRUCT
END_TYPE

// ---- Application/CSP/Main/Services/RFID FB/ST_BIS00LH_Outputs.TcDUT
TYPE ST_BIS00LH_Outputs :
STRUCT
	ByteArr AT %Q* : ARRAY[0..9] OF BYTE;
END_STRUCT
END_TYPE

// ---- Application/CSP/Main/Services/RFID FB/ST_BITHEADERIN.TcDUT
TYPE ST_BITHEADERIN :
STRUCT
	CP: BIT;
	AA: BIT;
	AE: BIT;
	AF: BIT;
	///unused
	Bit4: BIT;
	_TO: BIT;
	HF: BIT;
	BB: BIT;
END_STRUCT
END_TYPE

// ---- Application/CSP/Main/Services/RFID FB/ST_BITHEADEROUT.TcDUT
TYPE ST_BITHEADEROUT :
STRUCT
	AV: BIT;
	///unused
	Bit1: BIT;
	GR: BIT;
	///unused
	Bit3: BIT;
	///unused
	Bit4: BIT;
	KA: BIT;
	TI: BIT;
	///unused
	Bit7: BIT;
END_STRUCT
END_TYPE

// ---- Application/CSP/Transfer/Accumulator/csp_transfer_accumulator_belt_cam_enum.TcDUT
TYPE csp_transfer_accumulator_belt_cam_enum :
(
	IDLE							:= 33,
	RUN								:= 16	
);
END_TYPE

// ---- Application/CSP/Transfer/Accumulator/csp_transfer_accumulator_belt_connection_status_enum.TcDUT
TYPE csp_transfer_accumulator_belt_connection_status_enum :
(		
	CSP_TRANSFER_ACCUMULATOR_BELT_STATUS_CONNECTION_START					:= 0,
	CSP_TRANSFER_ACCUMULATOR_BELT_STATUS_CONNECTION_ENGAGE					:= 10,
	CSP_TRANSFER_ACCUMULATOR_BELT_STATUS_CONNECTION_ENGAGED					:= 20,
	CSP_TRANSFER_ACCUMULATOR_BELT_STATUS_CONNECTION_CHECK_CHANGE_CAM		:= 30,
	CSP_TRANSFER_ACCUMULATOR_BELT_STATUS_CONNECTION_CHANGE_CAM				:= 40,
	CSP_TRANSFER_ACCUMULATOR_BELT_STATUS_CONNECTION_WAIT_NEW_CAM			:= 50,
	CSP_TRANSFER_ACCUMULATOR_BELT_STATUS_CONNECTION_DONE 					:= 900,
	CSP_TRANSFER_ACCUMULATOR_BELT_STATUS_CONNECTION_ERROR 					:= 999
) := CSP_TRANSFER_ACCUMULATOR_BELT_STATUS_CONNECTION_START;
END_TYPE

// ---- Application/CSP/Transfer/Accumulator/csp_transfer_accumulator_belt_phase_status_enum.TcDUT
TYPE csp_transfer_accumulator_belt_phase_status_enum :
(		
	CSP_TRANSFER_ACCUMULATOR_BELT_STATUS_PHASE_START							:= 0,
	CSP_TRANSFER_ACCUMULATOR_BELT_STATUS_PHASE_DISABLE 							:= 10,
	CSP_TRANSFER_ACCUMULATOR_BELT_STATUS_PHASE_ENABLE 							:= 20,	
	CSP_TRANSFER_ACCUMULATOR_BELT_STATUS_PHASE_ENABLED 							:= 30,
	CSP_TRANSFER_ACCUMULATOR_BELT_STATUS_PHASE_CALCULATE_SLAVE_POSITION_REQUEST	:= 31,
	CSP_TRANSFER_ACCUMULATOR_BELT_STATUS_PHASE_CALCULATING_SLAVE_POSITION		:= 32,
	CSP_TRANSFER_ACCUMULATOR_BELT_STATUS_PHASE_REQUESTED						:= 33,
	CSP_TRANSFER_ACCUMULATOR_BELT_STATUS_PHASE_PHASING							:= 34,
	CSP_TRANSFER_ACCUMULATOR_BELT_STATUS_PHASE_PHASED							:= 35,
	CSP_TRANSFER_ACCUMULATOR_BELT_STATUS_PHASE_REDEFINE							:= 40,
	CSP_TRANSFER_ACCUMULATOR_BELT_STATUS_PHASE_REDEFINED						:= 50,
	CSP_TRANSFER_ACCUMULATOR_BELT_STATUS_PHASE_DONE 							:= 900,
	CSP_TRANSFER_ACCUMULATOR_BELT_STATUS_PHASE_ERROR 							:= 999
) := CSP_TRANSFER_ACCUMULATOR_BELT_STATUS_PHASE_START;
END_TYPE

// ---- Application/CSP/Transfer/Accumulator/csp_transfer_accumulator_belt_status_enum.TcDUT
TYPE csp_transfer_accumulator_belt_status_enum :
(
	CSP_TRANSFER_ACCUMULATOR_BELT_STATUS_NOT_INITIALIZED 							:=  0,
	CSP_TRANSFER_ACCUMULATOR_BELT_STATUS_DISABLED 									:=  10,
	CSP_TRANSFER_ACCUMULATOR_BELT_STATUS_ENABLE_REQUEST 							:=  20,
	CSP_TRANSFER_ACCUMULATOR_BELT_STATUS_ENABLING 									:=  30,
	CSP_TRANSFER_ACCUMULATOR_BELT_STATUS_ENABLED 									:=  40,
	CSP_TRANSFER_ACCUMULATOR_BELT_STATUS_HOME_REQUEST								:=  50,
	CSP_TRANSFER_ACCUMULATOR_BELT_STATUS_HOMING									:=  60,
	CSP_TRANSFER_ACCUMULATOR_BELT_STATUS_HOME_DONE									:=  70,
	CSP_TRANSFER_ACCUMULATOR_BELT_STATUS_CALCULATING_SLAVE_POSITION				:=  90,
	CSP_TRANSFER_ACCUMULATOR_BELT_STATUS_WAITING_SLAVE_ENGAGE						:= 100,
	CSP_TRANSFER_ACCUMULATOR_BELT_STATUS_PHASE_REQUEST								:= 140,
	CSP_TRANSFER_ACCUMULATOR_BELT_STATUS_PHASING									:= 150,
	CSP_TRANSFER_ACCUMULATOR_BELT_STATUS_PHASED									:= 160,
	CSP_TRANSFER_ACCUMULATOR_BELT_STATUS_CAM_ENGAGED_REQ							:= 170,
	CSP_TRANSFER_ACCUMULATOR_BELT_STATUS_AXIS_ENGAGE_VERIFY						:= 180,
	CSP_TRANSFER_ACCUMULATOR_BELT_STATUS_CAM_ENGAGED_EXTEND								:= 190,
	CSP_TRANSFER_ACCUMULATOR_BELT_STATUS_CAM_DISENAGE_WAIT							:= 191,
	CSP_TRANSFER_ACCUMULATOR_BELT_STATUS_CAM_ENGAGED_RETRACT							:= 192,
	CSP_TRANSFER_ACCUMULATOR_BELT_STATUS_CAM_TABLE_READ							:= 195,
	CSP_TRANSFER_ACCUMULATOR_BELT_STATUS_CALCULATE_SLAVE_POSITION_REQUEST			:= 196,
	CSP_TRANSFER_ACCUMULATOR_BELT_STATUS_READY										:= 197,
	CSP_TRANSFER_ACCUMULATOR_BELT_STATUS_RUNNING									:= 200,
	CSP_TRANSFER_ACCUMULATOR_BELT_STATUS_MOVING									:= 205,
	CSP_TRANSFER_ACCUMULATOR_BELT_STATUS_DISENGAGE_REQUEST						:= 210,
	CSP_TRANSFER_ACCUMULATOR_BELT_STATUS_DISENGAGING								:= 211,	
	CSP_TRANSFER_ACCUMULATOR_BELT_STATUS_REJECT									:= 220,
	CSP_TRANSFER_ACCUMULATOR_BELT_STATUS_REJECT_WAITING							:= 221,
	CSP_TRANSFER_ACCUMULATOR_BELT_STATUS_REJECT_COMPLETE							:= 222,
	CSP_TRANSFER_ACCUMULATOR_BELT_STATUS_STOP_REQUEST 								:= 500,
	CSP_TRANSFER_ACCUMULATOR_BELT_STATUS_DISABLE_REQUEST 							:= 530,
	CSP_TRANSFER_ACCUMULATOR_BELT_STATUS_DISABLING 								:= 540
) := CSP_TRANSFER_ACCUMULATOR_BELT_STATUS_NOT_INITIALIZED;
END_TYPE

// ---- Application/CSP/Transfer/Accumulator/csp_transfer_accumulator_connection_status_enum.TcDUT
TYPE csp_transfer_accumulator_connection_status_enum :
(		
	CSP_TRANSFER_ACCUMULATOR_STATUS_CONNECTION_START					:= 0,
	CSP_TRANSFER_ACCUMULATOR_STATUS_CONNECTION_ENGAGE					:= 10,
	CSP_TRANSFER_ACCUMULATOR_STATUS_CONNECTION_ENGAGED					:= 20,
	CSP_TRANSFER_ACCUMULATOR_STATUS_CONNECTION_CHECK_CHANGE_CAM			:= 30,
	CSP_TRANSFER_ACCUMULATOR_STATUS_CONNECTION_CHANGE_CAM				:= 40,
	CSP_TRANSFER_ACCUMULATOR_STATUS_CONNECTION_WAIT_NEW_CAM				:= 50,
	CSP_TRANSFER_ACCUMULATOR_STATUS_CONNECTION_DONE 					:= 900,
	CSP_TRANSFER_ACCUMULATOR_STATUS_CONNECTION_ERROR 					:= 999
) := CSP_TRANSFER_ACCUMULATOR_STATUS_CONNECTION_START;
END_TYPE

// ---- Application/CSP/Transfer/Accumulator/csp_transfer_accumulator_finger_status_enum.TcDUT
TYPE csp_transfer_accumulator_finger_status_enum :
(
	CSP_TRANSFER_ACCUMULATOR_FINGER_STATUS_NOT_INITIALIZED 							:=  0,
	CSP_TRANSFER_ACCUMULATOR_FINGER_STATUS_DISABLED 									:=  10,
	CSP_TRANSFER_ACCUMULATOR_FINGER_STATUS_ENABLE_REQUEST 							:=  20,
	CSP_TRANSFER_ACCUMULATOR_FINGER_STATUS_ENABLING 									:=  30,
	CSP_TRANSFER_ACCUMULATOR_FINGER_STATUS_ENABLED 									:=  40,
	CSP_TRANSFER_ACCUMULATOR_FINGER_STATUS_HOME_REQUEST								:=  50,
	CSP_TRANSFER_ACCUMULATOR_FINGER_STATUS_HOMING									:=  60,
	CSP_TRANSFER_ACCUMULATOR_FINGER_STATUS_HOME_DONE									:=  70,
	CSP_TRANSFER_ACCUMULATOR_FINGER_STATUS_CALCULATING_SLAVE_POSITION				:=  90,
	CSP_TRANSFER_ACCUMULATOR_FINGER_STATUS_WAITING_SLAVE_ENGAGE						:= 100,
	CSP_TRANSFER_ACCUMULATOR_FINGER_STATUS_PHASE_REQUEST								:= 140,
	CSP_TRANSFER_ACCUMULATOR_FINGER_STATUS_PHASING									:= 150,
	CSP_TRANSFER_ACCUMULATOR_FINGER_STATUS_PHASED									:= 160,
	CSP_TRANSFER_ACCUMULATOR_FINGER_STATUS_CAM_ENGAGED_REQ							:= 170,
	CSP_TRANSFER_ACCUMULATOR_FINGER_STATUS_AXIS_ENGAGE_VERIFY						:= 180,
	CSP_TRANSFER_ACCUMULATOR_FINGER_STATUS_CAM_ENGAGED								:= 190,
	CSP_TRANSFER_ACCUMULATOR_FINGER_STATUS_CAM_TABLE_READ							:= 195,
	CSP_TRANSFER_ACCUMULATOR_FINGER_STATUS_CALCULATE_SLAVE_POSITION_REQUEST			:= 196,
	CSP_TRANSFER_ACCUMULATOR_FINGER_STATUS_READY										:= 197,
	CSP_TRANSFER_ACCUMULATOR_FINGER_STATUS_RUNNING									:= 200,
	CSP_TRANSFER_ACCUMULATOR_FINGER_STATUS_MOVING									:= 205,
	CSP_TRANSFER_ACCUMULATOR_FINGER_STATUS_DISENGAGE_REQUEST						:= 210,
	CSP_TRANSFER_ACCUMULATOR_FINGER_STATUS_DISENGAGING								:= 211,	
	CSP_TRANSFER_ACCUMULATOR_FINGER_STATUS_STOP_REQUEST 								:= 500,
	CSP_TRANSFER_ACCUMULATOR_FINGER_STATUS_DISABLE_REQUEST 							:= 530,
	CSP_TRANSFER_ACCUMULATOR_FINGER_STATUS_DISABLING 								:= 540
) := CSP_TRANSFER_ACCUMULATOR_FINGER_STATUS_NOT_INITIALIZED;
END_TYPE

// ---- Application/CSP/Transfer/Accumulator/csp_transfer_accumulator_lift_status_enum.TcDUT
TYPE csp_transfer_accumulator_lift_status_enum :
(
	CSP_TRANSFER_ACCUMULATOR_LIFT_STATUS_NOT_INITIALIZED 							:=  0,
	CSP_TRANSFER_ACCUMULATOR_LIFT_STATUS_DISABLED 									:=  10,
	CSP_TRANSFER_ACCUMULATOR_LIFT_STATUS_ENABLE_REQUEST 							:=  20,
	CSP_TRANSFER_ACCUMULATOR_LIFT_STATUS_ENABLING 									:=  30,
	CSP_TRANSFER_ACCUMULATOR_LIFT_STATUS_ENABLED 									:=  40,
	CSP_TRANSFER_ACCUMULATOR_LIFT_STATUS_HOME_REQUEST								:=  50,
	CSP_TRANSFER_ACCUMULATOR_LIFT_STATUS_HOMING									:=  60,
	CSP_TRANSFER_ACCUMULATOR_LIFT_STATUS_HOME_DONE									:=  70,
	CSP_TRANSFER_ACCUMULATOR_LIFT_STATUS_CALCULATING_SLAVE_POSITION				:=  90,
	CSP_TRANSFER_ACCUMULATOR_LIFT_STATUS_WAITING_SLAVE_ENGAGE						:= 100,
	CSP_TRANSFER_ACCUMULATOR_LIFT_STATUS_PHASE_REQUEST								:= 140,
	CSP_TRANSFER_ACCUMULATOR_LIFT_STATUS_PHASING									:= 150,
	CSP_TRANSFER_ACCUMULATOR_LIFT_STATUS_PHASED									:= 160,
	CSP_TRANSFER_ACCUMULATOR_LIFT_STATUS_CAM_ENGAGED_REQ							:= 170,
	CSP_TRANSFER_ACCUMULATOR_LIFT_STATUS_AXIS_ENGAGE_VERIFY						:= 180,
	CSP_TRANSFER_ACCUMULATOR_LIFT_STATUS_CAM_ENGAGED								:= 190,
	CSP_TRANSFER_ACCUMULATOR_LIFT_STATUS_CAM_TABLE_READ							:= 195,
	CSP_TRANSFER_ACCUMULATOR_LIFT_STATUS_CALCULATE_SLAVE_POSITION_REQUEST			:= 196,
	CSP_TRANSFER_ACCUMULATOR_LIFT_STATUS_READY										:= 197,
	CSP_TRANSFER_ACCUMULATOR_LIFT_STATUS_RUNNING									:= 200,
	CSP_TRANSFER_ACCUMULATOR_LIFT_STATUS_MOVING									:= 205,
	CSP_TRANSFER_ACCUMULATOR_LIFT_STATUS_DISENGAGE_REQUEST						:= 210,
	CSP_TRANSFER_ACCUMULATOR_LIFT_STATUS_DISENGAGING								:= 211,	
	CSP_TRANSFER_ACCUMULATOR_LIFT_STATUS_STOP_REQUEST 								:= 500,
	CSP_TRANSFER_ACCUMULATOR_LIFT_STATUS_DISABLE_REQUEST 							:= 530,
	CSP_TRANSFER_ACCUMULATOR_LIFT_STATUS_DISABLING 								:= 540
) := CSP_TRANSFER_ACCUMULATOR_LIFT_STATUS_NOT_INITIALIZED;
END_TYPE

// ---- Application/CSP/Transfer/Crosspusher/csp_transfer_crosspusher_connection_status_enum.TcDUT
TYPE csp_transfer_crosspusher_connection_status_enum :
(		
	CSP_TRANSFER_CROSSPUSHER_STATUS_CONNECTION_START							:= 0,
	CSP_TRANSFER_CROSSPUSHER_STATUS_CONNECTION_ENGAGE							:= 10,
	CSP_TRANSFER_CROSSPUSHER_STATUS_CONNECTION_ENGAGED							:= 20,
	CSP_TRANSFER_CROSSPUSHER_STATUS_CONNECTION_CHECK_CHANGE_CAM					:= 30,
	CSP_TRANSFER_CROSSPUSHER_STATUS_CONNECTION_CHANGE_CAM						:= 40,
	CSP_TRANSFER_CROSSPUSHER_STATUS_CONNECTION_IMMEDIATE_CHANGE					:= 45,
	CSP_TRANSFER_CROSSPUSHER_STATUS_CONNECTION_WAIT_NEW_CAM						:= 50,
	CSP_TRANSFER_CROSSPUSHER_STATUS_CONNECTION_WAIT_REJECT						:= 60,
	CSP_TRANSFER_CROSSPUSHER_STATUS_CONNECTION_WAIT_REJECT_CAM_ENGAGE			:= 65,
	CSP_TRANSFER_CROSSPUSHER_STATUS_CONNECTION_DONE 							:= 900,
	CSP_TRANSFER_CROSSPUSHER_STATUS_CONNECTION_ERROR 							:= 999
) := CSP_TRANSFER_CROSSPUSHER_STATUS_CONNECTION_START;
END_TYPE

// ---- Application/CSP/Transfer/Crosspusher/csp_transfer_crosspusher_constant_struct.TcDUT
TYPE csp_transfer_crosspusher_constant_struct :
STRUCT
	(*BELT Info*)
	MIN_VELOCITY_MMpSEC:						LREAL := 100;
	MAX_VELOCITY_MMpSEC:						LREAL := 10000;
	MAX_ACCELERATION_MMpSEC2:					LREAL := 100000;
	MAX_DECELERATION_MMpSEC2:					LREAL := 100000;
	MAX_JERK_MMpSEC3:							LREAL := 1000000;
	RUNNING_ACCELERATION_MMMpSEC2:				LREAL := 30000;
	RUNNING_DECELERATION_MMpSEC2:				LREAL := 30000;
	MAX_FOLLOWING_ERROR_MM:						LREAL := 1000;
	
	RUNNING_JERK_MMpSEC3:						LREAL := 1000000;
	MOTOR_MAX_VELOCITY_DEGPS:					LREAL := 9600;
	MOTOR_MAX_ACCELERATION_DEGPS2:				LREAL := 4800;
	MOTOR_MAX_DECELERATION_DEGPS2:				LREAL := 4800;
	MOTOR_MAX_JERK_DEGPS3:						LREAL := 100000000; 
	MOTOR_MAX_FOLLOWING_ERROR_DEG:				LREAL := 2;
END_STRUCT
END_TYPE

// ---- Application/CSP/Transfer/Crosspusher/csp_transfer_crosspusher_follower_status_enum.TcDUT
TYPE csp_transfer_crosspusher_follower_status_enum :
(
	CSP_TRANSFER_CROSSPUSHER_FOLLOWER_STATUS_NOT_INITIALIZED 							:=  0,
	CSP_TRANSFER_CROSSPUSHER_FOLLOWER_STATUS_DISABLED 									:=  10,
	CSP_TRANSFER_CROSSPUSHER_FOLLOWER_STATUS_ENABLE_REQUEST 							:=  20,
	CSP_TRANSFER_CROSSPUSHER_FOLLOWER_STATUS_ENABLING 									:=  30,
	CSP_TRANSFER_CROSSPUSHER_FOLLOWER_STATUS_ENABLED 									:=  40,
	CSP_TRANSFER_CROSSPUSHER_FOLLOWER_STATUS_HOME_REQUEST								:=  50,
	CSP_TRANSFER_CROSSPUSHER_FOLLOWER_STATUS_HOMING										:=  60,
	CSP_TRANSFER_CROSSPUSHER_FOLLOWER_STATUS_HOME_DONE									:=  70,
	CSP_TRANSFER_CROSSPUSHER_FOLLOWER_STATUS_CALCULATING_SLAVE_POSITION					:=  90,
	CSP_TRANSFER_CROSSPUSHER_FOLLOWER_STATUS_WAITING_SLAVE_ENGAGE						:= 100,
	CSP_TRANSFER_CROSSPUSHER_FOLLOWER_STATUS_PHASE_REQUEST								:= 140,
	CSP_TRANSFER_CROSSPUSHER_FOLLOWER_STATUS_PHASING									:= 150,
	CSP_TRANSFER_CROSSPUSHER_FOLLOWER_STATUS_PHASED										:= 160,
	CSP_TRANSFER_CROSSPUSHER_FOLLOWER_STATUS_CAM_ENGAGED_REQ							:= 170,
	CSP_TRANSFER_CROSSPUSHER_FOLLOWER_STATUS_AXIS_ENGAGE_VERIFY							:= 180,
	CSP_TRANSFER_CROSSPUSHER_FOLLOWER_STATUS_CAM_ENGAGED_EXTEND							:= 190,
	CSP_TRANSFER_CROSSPUSHER_FOLLOWER_STATUS_CAM_DISENAGE_WAIT							:= 191,
	CSP_TRANSFER_CROSSPUSHER_FOLLOWER_STATUS_CAM_ENGAGED_RETRACT						:= 192,
	CSP_TRANSFER_CROSSPUSHER_FOLLOWER_STATUS_CAM_TABLE_READ								:= 195,
	CSP_TRANSFER_CROSSPUSHER_FOLLOWER_STATUS_CALCULATE_SLAVE_POSITION_REQUEST			:= 196,
	CSP_TRANSFER_CROSSPUSHER_FOLLOWER_STATUS_READY										:= 197,
	CSP_TRANSFER_CROSSPUSHER_FOLLOWER_STATUS_RUNNING									:= 200,
	CSP_TRANSFER_CROSSPUSHER_FOLLOWER_STATUS_MOVING										:= 205,
	CSP_TRANSFER_CROSSPUSHER_FOLLOWER_STATUS_DISENGAGE_REQUEST							:= 210,
	CSP_TRANSFER_CROSSPUSHER_FOLLOWER_STATUS_DISENGAGING								:= 211,	
	CSP_TRANSFER_CROSSPUSHER_FOLLOWER_STATUS_REJECT										:= 220,
	CSP_TRANSFER_CROSSPUSHER_FOLLOWER_STATUS_REJECT_WAITING								:= 221,
	CSP_TRANSFER_CROSSPUSHER_FOLLOWER_STATUS_REJECT_COMPLETE							:= 222,
	CSP_TRANSFER_CROSSPUSHER_FOLLOWER_STATUS_STOP_REQUEST 								:= 500,
	CSP_TRANSFER_CROSSPUSHER_FOLLOWER_STATUS_DISABLE_REQUEST 							:= 530,
	CSP_TRANSFER_CROSSPUSHER_FOLLOWER_STATUS_DISABLING 									:= 540
) := CSP_TRANSFER_CROSSPUSHER_FOLLOWER_STATUS_NOT_INITIALIZED;
END_TYPE

// ---- Application/CSP/Transfer/Crosspusher/csp_transfer_crosspusher_horizontal_constant_struct.TcDUT
TYPE csp_transfer_crosspusher_horizontal_constant_struct :
STRUCT
	(*BELT Info*)
	MIN_VELOCITY_MMpSEC:						LREAL := 100;
	MAX_VELOCITY_MMpSEC:						LREAL := 1000;
	MAX_ACCELERATION_MMpSEC2:					LREAL := 10000;
	MAX_DECELERATION_MMpSEC2:					LREAL := 10000;
	MAX_JERK_MMpSEC3:							LREAL := 1000000;
	RUNNING_ACCELERATION_MMMpSEC2:				LREAL := 3000;
	RUNNING_DECELERATION_MMpSEC2:				LREAL := 3000;
	MAX_FOLLOWING_ERROR_MM:						LREAL := 100;
	
	RUNNING_JERK_MMpSEC3:						LREAL := 1000000;
	MOTOR_MAX_VELOCITY_DEGPS:					LREAL := 9600;
	MOTOR_MAX_ACCELERATION_DEGPS2:				LREAL := 4800;
	MOTOR_MAX_DECELERATION_DEGPS2:				LREAL := 4800;
	MOTOR_MAX_JERK_DEGPS3:						LREAL := 100000000; 
	MOTOR_MAX_FOLLOWING_ERROR_DEG:				LREAL := 2;
END_STRUCT
END_TYPE

// ---- Application/CSP/Transfer/Crosspusher/csp_transfer_crosspusher_horizontal_status_enum.TcDUT
TYPE csp_transfer_crosspusher_horizontal_status_enum :
(
	CSP_TRANSFER_CROSSPUSHER_HORIZONTAL_STATUS_NOT_INITIALIZED 							:=  0,
	CSP_TRANSFER_CROSSPUSHER_HORIZONTAL_STATUS_DISABLED 								:=  10,
	CSP_TRANSFER_CROSSPUSHER_HORIZONTAL_STATUS_ENABLE_REQUEST 							:=  20,
	CSP_TRANSFER_CROSSPUSHER_HORIZONTAL_STATUS_ENABLING 								:=  30,
	CSP_TRANSFER_CROSSPUSHER_HORIZONTAL_STATUS_ENABLED 									:=  40,
	CSP_TRANSFER_CROSSPUSHER_HORIZONTAL_STATUS_HOME_REQUEST								:=  50,
	CSP_TRANSFER_CROSSPUSHER_HORIZONTAL_STATUS_HOMING									:=  60,
	CSP_TRANSFER_CROSSPUSHER_HORIZONTAL_STATUS_HOME_DONE								:=  70,
	CSP_TRANSFER_CROSSPUSHER_HORIZONTAL_STATUS_CALCULATE_SLAVE_POSITION_REQUEST			:= 80,
	CSP_TRANSFER_CROSSPUSHER_HORIZONTAL_STATUS_CALCULATING_SLAVE_POSITION				:= 90,
	CSP_TRANSFER_CROSSPUSHER_HORIZONTAL_STATUS_WAITING_SLAVE_ENGAGE						:= 100,
	CSP_TRANSFER_CROSSPUSHER_HORIZONTAL_STATUS_PHASE_REQUEST							:= 140,
	CSP_TRANSFER_CROSSPUSHER_HORIZONTAL_STATUS_PHASING									:= 150,
	CSP_TRANSFER_CROSSPUSHER_HORIZONTAL_STATUS_PHASED									:= 160,
	CSP_TRANSFER_CROSSPUSHER_HORIZONTAL_STATUS_CAM_ENGAGED_REQ							:= 170,
	CSP_TRANSFER_CROSSPUSHER_HORIZONTAL_STATUS_AXIS_ENGAGE_VERIFY						:= 180,
	CSP_TRANSFER_CROSSPUSHER_HORIZONTAL_STATUS_CAM_ENGAGED								:= 190,
	CSP_TRANSFER_CROSSPUSHER_HORIZONTAL_STATUS_CAM_TABLE_READ							:= 195,
	CSP_TRANSFER_CROSSPUSHER_HORIZONTAL_STATUS_READY									:= 197,
	CSP_TRANSFER_CROSSPUSHER_HORIZONTAL_STATUS_RUNNING									:= 200,
	CSP_TRANSFER_CROSSPUSHER_HORIZONTAL_STATUS_MOVING									:= 205,
	CSP_TRANSFER_CROSSPUSHER_HORIZONTAL_STATUS_DISENGAGE_REQUEST						:= 210,
	CSP_TRANSFER_CROSSPUSHER_HORIZONTAL_STATUS_DISENGAGING								:= 211,	
	CSP_TRANSFER_CROSSPUSHER_HORIZONTAL_STATUS_REJECT									:= 220,
	CSP_TRANSFER_CROSSPUSHER_HORIZONTAL_STATUS_REJECT_WAITING							:= 221,
	CSP_TRANSFER_CROSSPUSHER_HORIZONTAL_STATUS_REJECT_COMPLETE							:= 222,
	CSP_TRANSFER_CROSSPUSHER_HORIZONTAL_STATUS_STOP_REQUEST 							:= 500,
	CSP_TRANSFER_CROSSPUSHER_HORIZONTAL_STATUS_DISABLE_REQUEST 							:= 530,
	CSP_TRANSFER_CROSSPUSHER_HORIZONTAL_STATUS_DISABLING 								:= 540
) := CSP_TRANSFER_CROSSPUSHER_HORIZONTAL_STATUS_NOT_INITIALIZED;
END_TYPE

// ---- Application/CSP/Transfer/Crosspusher/csp_transfer_crosspusher_loader_clear_status.TcDUT
TYPE csp_transfer_crosspusher_loader_clear_status :
(
	NONE							:= 0,
	NOT_CLEAR						:= 1,
	CLEAR							:= 2	
);
END_TYPE

// ---- Application/CSP/Transfer/Crosspusher/csp_transfer_crosspusher_phase_status_enum.TcDUT
TYPE csp_transfer_crosspusher_phase_status_enum :
(		
	CSP_TRANSFER_CROSSPUSHER_PHASE_STATUS_START									:= 0,
	CSP_TRANSFER_CROSSPUSHER_PHASE_STATUS_DISABLE 								:= 10,
	CSP_TRANSFER_CROSSPUSHER_PHASE_STATUS_ENABLE 								:= 20,	
	CSP_TRANSFER_CROSSPUSHER_PHASE_STATUS_ENABLED 								:= 30,
	CSP_TRANSFER_CROSSPUSHER_PHASE_STATUS_CALCULATE_SLAVE_POSITION_REQUEST		:= 31,
	CSP_TRANSFER_CROSSPUSHER_PHASE_STATUS_CALCULATING_SLAVE_POSITION			:= 32,
	CSP_TRANSFER_CROSSPUSHER_PHASE_PHASE_STATUS_REQUEST							:= 33,
	CSP_TRANSFER_CROSSPUSHER_PHASE_STATUS_PHASING								:= 34,
	CSP_TRANSFER_CROSSPUSHER_PHASE_STATUS_PHASED								:= 35,
	CSP_TRANSFER_CROSSPUSHER_PHASE_STATUS_REDEFINE								:= 40,
	CSP_TRANSFER_CROSSPUSHER_PHASE_STATUS_REDEFINED								:= 50,
	CSP_TRANSFER_CROSSPUSHER_PHASE_STATUS_CHECK_STACK_COUNT						:= 100,
	CSP_TRANSFER_CROSSPUSHER_PHASE_STATUS_CHECK_IF_LIFT_VERT					:= 105,
	CSP_TRANSFER_CROSSPUSHER_PHASE_STATUS_DISABLE_VERTICAL						:= 110,
	CSP_TRANSFER_CROSSPUSHER_PHASE_STATUS_ENABLE_VERTICAL						:= 120,
	CSP_TRANSFER_CROSSPUSHER_PHASE_STATUS_LIFT_VERTICAL							:= 130,
	CSP_TRANSFER_CROSSPUSHER_PHASE_STATUS_VERTICAL_LIFTING						:= 140,
	CSP_TRANSFER_CROSSPUSHER_PHASE_STATUS_VERTICAL_LIFTED						:= 150,
	CSP_TRANSFER_CROSSPUSHER_PHASE_STATUS_NOT_POSSIBLE							:= 800,
	CSP_TRANSFER_CROSSPUSHER_PHASE_STATUS_DONE 									:= 900,
	CSP_TRANSFER_CROSSPUSHER_PHASE_STATUS_ERROR 								:= 999
) := CSP_TRANSFER_CROSSPUSHER_PHASE_STATUS_START;
END_TYPE

// ---- Application/CSP/Transfer/Crosspusher/csp_transfer_crosspusher_reject_status_enum.TcDUT
TYPE csp_transfer_crosspusher_reject_status_enum :
(		
	CSP_TRANSFER_CROSSPUSHER_REJECT_STATUS_START							:= 0,
	CSP_TRANSFER_CROSSPUSHER_REJECT_STATUS_DWELL_TRANSFER_VM				:= 5,
	CSP_TRANSFER_CROSSPUSHER_REJECT_STATUS_DISENGAGE_AXES					:= 20,
	CSP_TRANSFER_CROSSPUSHER_REJECT_STATUS_GEAR_FOLLOWER					:= 30,
	CSP_TRANSFER_CROSSPUSHER_REJECT_STATUS_MOVE_TO_REJECT_POS				:= 40,
	CSP_TRANSFER_CROSSPUSHER_REJECT_STATUS_VERIFY_HORIZONTAL_POS			:= 50,
	CSP_TRANSFER_CROSSPUSHER_REJECT_STATUS_UNGEAR_FOLLOWER					:= 51,
	CSP_TRANSFER_CROSSPUSHER_REJECT_STATUS_MOVE_FOLLOWER					:= 52,
	CSP_TRANSFER_CROSSPUSHER_REJECT_STATUS_VERIFY_FOLLOWER_POS				:= 53,
	CSP_TRANSFER_CROSSPUSHER_REJECT_STATUS_REJECT_STACK 					:= 60,
	CSP_TRANSFER_CROSSPUSHER_REJECT_STATUS_VERIFY							:= 80,
	CSP_TRANSFER_CROSSPUSHER_REJECT_STATUS_RETURN_HORIZONTAL				:= 90,
	CSP_TRANSFER_CROSSPUSHER_REJECT_STATUS_HORIZONTAL_RETURNING				:= 91,
	CSP_TRANSFER_CROSSPUSHER_REJECT_STATUS_RETURN_FOLLOWER					:= 92,
	CSP_TRANSFER_CROSSPUSHER_REJECT_STATUS_FOLLOWER_RETURNING				:= 93,
	CSP_TRANSFER_CROSSPUSHER_REJECT_STATUS_VERIFY_AT_LOAD					:= 95,
	CSP_TRANSFER_CROSSPUSHER_REJECT_STATUS_RUN_AXES							:= 100, 
	CSP_TRANSFER_CROSSPUSHER_REJECT_STATUS_DONE								:= 120,
	CSP_TRANSFER_CROSSPUSHER_REJECT_STATUS_WAITING							:= 130,
	CSP_TRANSFER_CROSSPUSHER_REJECT_STATUS_EMERGENCY_STOP					:= 150,
	CSP_TRANSFER_CROSSPUSHER_REJECT_STATUS_EMERGENCY_STOP_ENABLE			:= 160,
	CSP_TRANSFER_CROSSPUSHER_REJECT_STATUS_EMERGENCY_STOP_GOTO				:= 170,
	CSP_TRANSFER_CROSSPUSHER_REJECT_STATUS_EMERGENCY_STOP_FOLLOWER_MOVE		:= 180
) := CSP_TRANSFER_CROSSPUSHER_REJECT_STATUS_START;
END_TYPE

// ---- Application/CSP/Transfer/Crosspusher/csp_transfer_crosspusher_status_enum.TcDUT
TYPE csp_transfer_crosspusher_status_enum :
(
	CSP_TRANSFER_CROSSPUSHER_STATUS_NOT_INITIALIZED 						:= 0,
	CSP_TRANSFER_CROSSPUSHER_STATUS_DISABLED 								:= 10,
	CSP_TRANSFER_CROSSPUSHER_STATUS_ENABLE_REQUEST 							:= 20,
	CSP_TRANSFER_CROSSPUSHER_STATUS_ENABLING 								:= 30,
	CSP_TRANSFER_CROSSPUSHER_STATUS_ENABLED 								:= 40,
	CSP_TRANSFER_CROSSPUSHER_STATUS_HOME_REQUEST							:= 50,
	CSP_TRANSFER_CROSSPUSHER_STATUS_HOMING									:= 60,
	CSP_TRANSFER_CROSSPUSHER_STATUS_HOME_DONE								:= 70,
	CSP_TRANSFER_CROSSPUSHER_STATUS_CALCULATE_SLAVE_POSITION_REQUEST		:= 80,
	CSP_TRANSFER_CROSSPUSHER_STATUS_CALCULATING_SLAVE_POSITION				:= 90,
	CSP_TRANSFER_CROSSPUSHER_STATUS_PHASE_REQUEST							:= 140,
	CSP_TRANSFER_CROSSPUSHER_STATUS_PHASING									:= 150,
	CSP_TRANSFER_CROSSPUSHER_STATUS_PHASED									:= 160,
	CSP_TRANSFER_CROSSPUSHER_STATUS_CAM_ENGAGED_REQ							:= 170,
	CSP_TRANSFER_CROSSPUSHER_STATUS_AXIS_ENGAGE_VERIFY						:= 180,
	CSP_TRANSFER_CROSSPUSHER_STATUS_CAM_ENGAGED								:= 190,
	CSP_TRANSFER_CROSSPUSHER_STATUS_CAM_TABLE_READ							:= 195,
	CSP_TRANSFER_CROSSPUSHER_STATUS_RUNNING									:= 200,
	CSP_TRANSFER_CROSSPUSHER_STATUS_REJECT									:= 205,
	CSP_TRANSFER_CROSSPUSHER_STATUS_CAM_DISENGAGE							:= 210,
	CSP_TRANSFER_CROSSPUSHER_STATUS_CAM_DISENGAGED							:= 220,
	CSP_TRANSFER_CROSSPUSHER_STATUS_CAM_UPDATING							:= 230,
	CSP_TRANSFER_CROSSPUSHER_STATUS_STOP_REQUEST 							:= 500,
	CSP_TRANSFER_CROSSPUSHER_STATUS_DISABLE_REQUEST 						:= 530,
	CSP_TRANSFER_CROSSPUSHER_STATUS_DISABLING 								:= 540
) := CSP_TRANSFER_CROSSPUSHER_STATUS_NOT_INITIALIZED;
END_TYPE

// ---- Application/CSP/Transfer/Crosspusher/csp_transfer_crosspusher_vertical_status_enum.TcDUT
TYPE csp_transfer_crosspusher_vertical_status_enum :
(
	CSP_TRANSFER_CROSSPUSHER_VERTICAL_STATUS_NOT_INITIALIZED 							:=  0,
	CSP_TRANSFER_CROSSPUSHER_VERTICAL_STATUS_DISABLED 									:=  10,
	CSP_TRANSFER_CROSSPUSHER_VERTICAL_STATUS_ENABLE_REQUEST 							:=  20,
	CSP_TRANSFER_CROSSPUSHER_VERTICAL_STATUS_ENABLING 									:=  30,
	CSP_TRANSFER_CROSSPUSHER_VERTICAL_STATUS_ENABLED 									:=  40,
	CSP_TRANSFER_CROSSPUSHER_VERTICAL_STATUS_HOME_REQUEST								:=  50,
	CSP_TRANSFER_CROSSPUSHER_VERTICAL_STATUS_HOMING										:=  60,
	CSP_TRANSFER_CROSSPUSHER_VERTICAL_STATUS_HOME_DONE									:=  70,
	CSP_TRANSFER_CROSSPUSHER_VERTICAL_STATUS_CALCULATE_SLAVE_POSITION_REQUEST			:=  80,
	CSP_TRANSFER_CROSSPUSHER_VERTICAL_STATUS_CALCULATING_SLAVE_POSITION					:=  90,
	CSP_TRANSFER_CROSSPUSHER_VERTICAL_STATUS_WAITING_SLAVE_ENGAGE						:= 100,
	CSP_TRANSFER_CROSSPUSHER_VERTICAL_STATUS_PHASE_REQUEST								:= 140,
	CSP_TRANSFER_CROSSPUSHER_VERTICAL_STATUS_PHASING									:= 150,
	CSP_TRANSFER_CROSSPUSHER_VERTICAL_STATUS_PHASED										:= 160,
	CSP_TRANSFER_CROSSPUSHER_VERTICAL_STATUS_CAM_ENGAGED_REQ							:= 170,
	CSP_TRANSFER_CROSSPUSHER_VERTICAL_STATUS_AXIS_ENGAGE_VERIFY							:= 180,
	CSP_TRANSFER_CROSSPUSHER_VERTICAL_STATUS_CAM_ENGAGED								:= 190,
	CSP_TRANSFER_CROSSPUSHER_VERTICAL_STATUS_CAM_TABLE_READ								:= 195,
	CSP_TRANSFER_CROSSPUSHER_VERTICAL_STATUS_READY										:= 197,
	CSP_TRANSFER_CROSSPUSHER_VERTICAL_STATUS_RUNNING									:= 200,
	CSP_TRANSFER_CROSSPUSHER_VERTICAL_STATUS_MOVING										:= 205,
	CSP_TRANSFER_CROSSPUSHER_VERTICAL_STATUS_DISENGAGE_REQUEST							:= 210,
	CSP_TRANSFER_CROSSPUSHER_VERTICAL_STATUS_DISENGAGING								:= 211,	
	CSP_TRANSFER_CROSSPUSHER_VERTICAL_STATUS_REJECT										:= 220,
	CSP_TRANSFER_CROSSPUSHER_VERTICAL_STATUS_REJECT_WAITING								:= 221,
	CSP_TRANSFER_CROSSPUSHER_VERTICAL_STATUS_REJECT_COMPLETE							:= 222,
	CSP_TRANSFER_CROSSPUSHER_VERTICAL_STATUS_STOP_REQUEST 								:= 500,
	CSP_TRANSFER_CROSSPUSHER_VERTICAL_STATUS_DISABLE_REQUEST 							:= 530,
	CSP_TRANSFER_CROSSPUSHER_VERTICAL_STATUS_DISABLING 									:= 540
) := CSP_TRANSFER_CROSSPUSHER_VERTICAL_STATUS_NOT_INITIALIZED;
END_TYPE

// ---- Application/CSP/Transfer/csp_transfer_connection_status_enum.TcDUT
TYPE csp_transfer_connection_status_enum :
(		
	CSP_TRANSFER_STATUS_CONNECTION_START							:= 0,
	CSP_TRANSFER_STATUS_CONNECTION_ENGAGE							:= 10,
	CSP_TRANSFER_STATUS_CONNECTION_ENGAGED						:= 20,
	CSP_TRANSFER_STATUS_CONNECTION_CHECK_CHANGE_CAM				:= 30,
	CSP_TRANSFER_STATUS_CONNECTION_CHANGE_CAM						:= 40,
	CSP_TRANSFER_STATUS_CONNECTION_WAIT_NEW_CAM					:= 50,
	CSP_TRANSFER_STATUS_CONNECTION_DONE 							:= 900,
	CSP_TRANSFER_STATUS_CONNECTION_ERROR 							:= 999
) := CSP_TRANSFER_STATUS_CONNECTION_START;
END_TYPE

// ---- Application/CSP/Transfer/csp_transfer_phase_status_enum.TcDUT
TYPE csp_transfer_phase_status_enum :
(		
	CSP_TRANSFER_PHASE_STATUS_START									:= 0,
	CSP_TRANSFER_PHASE_STATUS_DISABLE 								:= 10,
	CSP_TRANSFER_PHASE_STATUS_ENABLE 								:= 20,	
	CSP_TRANSFER_PHASE_STATUS_ENABLED 								:= 30,
	CSP_TRANSFER_PHASE_STATUS_CALCULATE_SLAVE_POSITION_REQUEST		:= 31,
	CSP_TRANSFER_PHASE_STATUS_CALCULATING_SLAVE_POSITION			:= 32,
	CSP_TRANSFER_PHASE_STATUS_REQUEST								:= 33,
	CSP_TRANSFER_PHASE_STATUS_PHASING								:= 34,
	CSP_TRANSFER_PHASE_STATUS_PHASED								:= 35,
	CSP_TRANSFER_PHASE_STATUS_REDEFINE								:= 40,
	CSP_TRANSFER_PHASE_STATUS_REDEFINED								:= 50,
	CSP_TRANSFER_PHASE_STATUS_DONE 									:= 900,
	CSP_TRANSFER_PHASE_STATUS_ERROR 								:= 999
) := CSP_TRANSFER_PHASE_STATUS_START;
END_TYPE

// ---- Application/CSP/Transfer/csp_transfer_status_enum.TcDUT
TYPE csp_transfer_status_enum :
(
	CSP_TRANSFER_STATUS_NOT_INITIALIZED 						:= 0,
	CSP_TRANSFER_STATUS_DISABLED 								:= 10,
	CSP_TRANSFER_STATUS_ENABLE_REQUEST 							:= 20,
	CSP_TRANSFER_STATUS_ENABLING 								:= 30,
	CSP_TRANSFER_STATUS_ENABLED 								:= 40,
	CSP_TRANSFER_STATUS_HOME_REQUEST							:= 50,
	CSP_TRANSFER_STATUS_HOMING									:= 60,
	CSP_TRANSFER_STATUS_HOME_DONE								:= 70,
	CSP_TRANSFER_STATUS_CALCULATE_SLAVE_POSITION_REQUEST		:= 80,
	CSP_TRANSFER_STATUS_CALCULATING_SLAVE_POSITION				:= 90,
	CSP_TRANSFER_STATUS_PHASE_REQUEST							:= 140,
	CSP_TRANSFER_STATUS_PHASING									:= 150,
	CSP_TRANSFER_STATUS_PHASED									:= 160,
	CSP_TRANSFER_STATUS_CAM_ENGAGED_REQ							:= 170,
	CSP_TRANSFER_STATUS_AXIS_ENGAGE_VERIFY						:= 180,
	CSP_TRANSFER_STATUS_CAM_ENGAGED								:= 190,
	CSP_TRANSFER_STATUS_CAM_CHANGE								:= 192,
	CSP_TRANSFER_STATUS_CAM_TABLE_READ							:= 195,
	CSP_TRANSFER_STATUS_RUNNING									:= 200,
	CSP_TRANSFER_STATUS_CAM_DISENGAGE							:= 210,
	CSP_TRANSFER_STATUS_CAM_DISENGAGED							:= 220,
	CSP_TRANSFER_STATUS_CAM_UPDATING							:= 230,
	CSP_TRANSFER_STATUS_REJECT									:= 250,
	CSP_TRANSFER_STATUS_STOP_REQUEST 							:= 500,
	CSP_TRANSFER_STATUS_DISABLE_REQUEST 						:= 530,
	CSP_TRANSFER_STATUS_DISABLING 								:= 540
) := CSP_TRANSFER_STATUS_NOT_INITIALIZED;
END_TYPE

// ---- Application/CSP/Transfer/Infeed/csp_transfer_infeed_belt_status_enum.TcDUT
TYPE csp_transfer_infeed_belt_status_enum :(
	CSP_TRANSFER_INFEED_BELT_STATUS_NOT_INITIALIZED 							:= 0,
	CSP_TRANSFER_INFEED_BELT_STATUS_DISABLED 									:= 10,
	CSP_TRANSFER_INFEED_BELT_STATUS_ENABLE_REQUEST 								:= 70,
	CSP_TRANSFER_INFEED_BELT_STATUS_ENABLING 									:= 80,
	CSP_TRANSFER_INFEED_BELT_STATUS_ENABLED 									:= 100,
	CSP_TRANSFER_INFEED_BELT_STATUS_RUNNING										:= 110,
	CSP_TRANSFER_INFEED_BELT_STATUS_STOP_REQUEST 								:= 500,
	CSP_TRANSFER_INFEED_BELT_STATUS_DISABLE_REQUEST 							:= 530,
	CSP_TRANSFER_INFEED_BELT_STATUS_DISABLING 									:= 540
	) := CSP_TRANSFER_INFEED_BELT_STATUS_NOT_INITIALIZED;
END_TYPE

// ---- Application/CSP/Transfer/Infeed/csp_transfer_infeed_connection_status_enum.TcDUT
TYPE csp_transfer_infeed_connection_status_enum :
(		
	CSP_TRANSFER_INFEED_STATUS_CONNECTION_START							:= 0,
	CSP_TRANSFER_INFEED_STATUS_CONNECTION_ENGAGE							:= 10,
	CSP_TRANSFER_INFEED_STATUS_CONNECTION_ENGAGED						:= 20,
	CSP_TRANSFER_INFEED_STATUS_CONNECTION_CHECK_CHANGE_CAM				:= 30,
	CSP_TRANSFER_INFEED_STATUS_CONNECTION_CHANGE_CAM						:= 40,
	CSP_TRANSFER_INFEED_STATUS_CONNECTION_WAIT_NEW_CAM					:= 50,
	CSP_TRANSFER_INFEED_STATUS_CONNECTION_DONE 							:= 900,
	CSP_TRANSFER_INFEED_STATUS_CONNECTION_ERROR 							:= 999
) := CSP_TRANSFER_INFEED_STATUS_CONNECTION_START;
END_TYPE

// ---- Application/CSP/Transfer/Infeed/csp_transfer_infeed_constant_struct.TcDUT
TYPE csp_transfer_infeed_constant_struct :
STRUCT
	(*BELT Info*)
	MIN_VELOCITY_HZ:							LREAL := 0;
	MAX_VELOCITY_HZ:							LREAL := 15000;
	MAX_ACCELERATION_HZpSEC:					LREAL := 2500;
	MAX_DECELERATION_HZpSEC:					LREAL := 2500;
	MAX_JERK_HZpSEC2:							LREAL := 25000;
	RUNNING_ACCELERATION_MMMpSEC2:				LREAL := 2500;
	RUNNING_DECELERATION_MMpSEC2:				LREAL := 2500;
	MAX_FOLLOWING_ERROR_MM:						LREAL := 100;
	
	RUNNING_JERK_MMpSEC3:						LREAL := 1000000;
	MOTOR_MAX_VELOCITY_DEGPS:					LREAL := 9600;
	MOTOR_MAX_ACCELERATION_DEGPS2:				LREAL := 4800;
	MOTOR_MAX_DECELERATION_DEGPS2:				LREAL := 4800;
	MOTOR_MAX_JERK_DEGPS3:						LREAL := 100000000; 
	MOTOR_MAX_FOLLOWING_ERROR_DEG:				LREAL := 2;
END_STRUCT
END_TYPE

// ---- Application/CSP/Transfer/Upstacker/csp_transfer_upstacker_carton_backstop.TcDUT
TYPE csp_transfer_upstacker_carton_backstop :
STRUCT
	status: 					csp_transfer_upstacker_carton_backstop_status;	
	change_cam_phase:			LREAL;	
END_STRUCT
END_TYPE

// ---- Application/CSP/Transfer/Upstacker/csp_transfer_upstacker_carton_backstop_status.TcDUT
TYPE csp_transfer_upstacker_carton_backstop_status :
(
	NONE							:= 0,
	PRESENT							:= 1,
	ABSENT							:= 2	
);
END_TYPE

// ---- Application/CSP/Transfer/Upstacker/csp_transfer_upstacker_connection_status_enum.TcDUT
TYPE csp_transfer_upstacker_connection_status_enum :
(		
	CSP_TRANSFER_UPSTACKER_STATUS_CONNECTION_START							:= 0,
	CSP_TRANSFER_UPSTACKER_STATUS_CONNECTION_ENGAGE							:= 10,
	CSP_TRANSFER_UPSTACKER_STATUS_CONNECTION_ENGAGED						:= 20,
	CSP_TRANSFER_UPSTACKER_STATUS_CONNECTION_CHECK_CHANGE_CAM				:= 30,
	CSP_TRANSFER_UPSTACKER_STATUS_CONNECTION_CHANGE_CAM						:= 40,
	CSP_TRANSFER_UPSTACKER_STATUS_CONNECTION_WAIT_NEW_CAM					:= 50,
	CSP_TRANSFER_UPSTACKER_STATUS_CONNECTION_DONE 							:= 900,
	CSP_TRANSFER_UPSTACKER_STATUS_CONNECTION_ERROR 							:= 999
) := CSP_TRANSFER_UPSTACKER_STATUS_CONNECTION_START;
END_TYPE

// ---- Application/CSP/Transfer/Upstacker/csp_transfer_upstacker_constant_struct.TcDUT
TYPE csp_transfer_upstacker_constant_struct :
STRUCT
	(*BELT Info*)
	MIN_VELOCITY_MMpSEC:						LREAL := 100;
	MAX_VELOCITY_MMpSEC:						LREAL := 1000;
	MAX_ACCELERATION_MMpSEC2:					LREAL := 10000;
	MAX_DECELERATION_MMpSEC2:					LREAL := 10000;
	MAX_JERK_MMpSEC3:							LREAL := 1000000;
	RUNNING_ACCELERATION_MMMpSEC2:				LREAL := 3000;
	RUNNING_DECELERATION_MMpSEC2:				LREAL := 3000;
	MAX_FOLLOWING_ERROR_MM:						LREAL := 100;
	
	RUNNING_JERK_MMpSEC3:						LREAL := 1000000;
	MOTOR_MAX_VELOCITY_DEGPS:					LREAL := 9600;
	MOTOR_MAX_ACCELERATION_DEGPS2:				LREAL := 4800;
	MOTOR_MAX_DECELERATION_DEGPS2:				LREAL := 4800;
	MOTOR_MAX_JERK_DEGPS3:						LREAL := 100000000; 
	MOTOR_MAX_FOLLOWING_ERROR_DEG:				LREAL := 2;
END_STRUCT
END_TYPE

// ---- Application/CSP/Transfer/Upstacker/csp_transfer_upstacker_phase_status_enum.TcDUT
TYPE csp_transfer_upstacker_phase_status_enum :
(		
	CSP_TRANSFER_UPSTACKER_STATUS_PHASE_START								:= 0,
	CSP_TRANSFER_UPSTACKER_STATUS_PHASE_CHECK_VM_STATUS						:= 1,
	CSP_TRANSFER_UPSTACKER_STATUS_PHASE_GET_VM_POS							:= 2,
	CSP_TRANSFER_UPSTACKER_STATUS_PHASE_CALCULATE_SLAVE_POS					:= 3,
	CSP_TRANSFER_UPSTACKER_STATUS_PHASE_CALCULATE_SLAVE_DOWN_POS			:= 600,
	CSP_TRANSFER_UPSTACKER_STATUS_PHASE_CHECK_CALCULATED_SLAVE_DOWN_POS		:= 601,
	CSP_TRANSFER_UPSTACKER_STATUS_PHASE_CALCULATE_SLAVE_UP_POS				:= 602,
	CSP_TRANSFER_UPSTACKER_STATUS_PHASE_CHECK_CALCULATED_SLAVE_UP_POS		:= 603,
	CSP_TRANSFER_UPSTACKER_STATUS_PHASE_CALCULATE_SLAVE_LS_FINGER_POS		:= 604,
	CSP_TRANSFER_UPSTACKER_STATUS_PHASE_CHECK_CALCULATED_SLAVE_LSFINGR_POS	:= 605,
	CSP_TRANSFER_UPSTACKER_STATUS_PHASE_CALCULATE_SLAVE_OS_FINGER_POS		:= 606,
	CSP_TRANSFER_UPSTACKER_STATUS_PHASE_CHECK_CALCULATED_SLAVE_OSFINGR_POS	:= 607,
	CSP_TRANSFER_UPSTACKER_STATUS_PHASE_CHECK_SLAVE_POS						:= 4,
	CSP_TRANSFER_UPSTACKER_STATUS_PHASE_SIMPLE_MOVE_AVAILABLE				:= 5,
	CSP_TRANSFER_UPSTACKER_STATUS_PHASE_CALCULATE_IDLE_POSITION				:= 10,
	CSP_TRANSFER_UPSTACKER_STATUS_PHASE_REDEFINE_IDLE_POSITION				:= 15,
	CSP_TRANSFER_UPSTACKER_STATUS_PHASE_READ_IDLE_POSITION					:= 20,
	CSP_TRANSFER_UPSTACKER_STATUS_PHASE_CALCULATE_SLAVE_POSITION			:= 30,
	CSP_TRANSFER_UPSTACKER_STATUS_PHASE_READ_SLAVE_POSITION					:= 40,
	CSP_TRANSFER_UPSTACKER_STATUS_PHASE_CALCULATE_VIRTUAL_POSITION			:= 50,
	CSP_TRANSFER_UPSTACKER_STATUS_PHASE_READ_VIRTUAL_POSITION				:= 60,
	CSP_TRANSFER_UPSTACKER_STATUS_PHASE_CHECK_CASE							:= 70,
	CSP_TRANSFER_UPSTACKER_STATUS_PHASE_DISABLE 							:= 80,
	CSP_TRANSFER_UPSTACKER_STATUS_PHASE_ENABLE 								:= 90,
	CSP_TRANSFER_UPSTACKER_STATUS_PHASE_ENABLED								:= 100,
	CSP_TRANSFER_UPSTACKER_STATUS_PHASE_CHECK_UPSTREAM_SKIP_PHASING			:= 101,
	CSP_TRANSFER_UPSTACKER_STATUS_PHASE_CHECK_DOWNSTREAM_SKIP_PHASE_1		:= 110,
	CSP_TRANSFER_UPSTACKER_STATUS_PHASE_CALCULATE_MASTER_POSITION			:= 150,
	CSP_TRANSFER_UPSTACKER_STATUS_PHASE_READ_MASTER_POSITION				:= 160,
	CSP_TRANSFER_UPSTACKER_STATUS_PHASE_ERROR_ON_MASTER_CALC				:= 161,
	CSP_TRANSFER_UPSTACKER_STATUS_PHASE_MOVE_UPSTREAM_FROM_ERROR_POS		:= 162,
	CSP_TRANSFER_UPSTACKER_STATUS_PHASE_WAIT_MOVE_DONE_UP_FROM_ERROR_POS	:= 163,
	CSP_TRANSFER_UPSTACKER_STATUS_PHASE_MOVE_DOWNSTREAM_FROM_ERROR_POS		:= 164,
	CSP_TRANSFER_UPSTACKER_STATUS_PHASE_WAIT_MOVE_DONE_DOWN_FROM_ERROR_POS	:= 165,
	CSP_TRANSFER_UPSTACKER_STATUS_PHASE_REDEFINE_MASTER_POSITION_STEP1		:= 170,
	CSP_TRANSFER_UPSTACKER_STATUS_PHASE_ENGAGE_DOWNSTREAM_STEP1				:= 180,
	CSP_TRANSFER_UPSTACKER_STATUS_PHASE_ENGAGE_UPSTREAM_STEP1				:= 190,
	CSP_TRANSFER_UPSTACKER_STATUS_PHASE_MOVE_MASTER_STEP1					:= 200,
	CSP_TRANSFER_UPSTACKER_STATUS_PHASE_DISENGAGE_STEP1						:= 210,
	CSP_TRANSFER_UPSTACKER_STATUS_PHASE_DISENGAGED_STEP1					:= 220,
	CSP_TRANSFER_UPSTACKER_STATUS_PHASE_CALCULE_DOWNSTREAM_START_POSITION_1	:= 230,
	CSP_TRANSFER_UPSTACKER_STATUS_PHASE_MOVE_DOWNSTREAM_START_POSITION_1	:= 240,
	CSP_TRANSFER_UPSTACKER_STATUS_PHASE_MOVED_DOWNSTREAM_START_POSITION_1	:= 250,
	CSP_TRANSFER_UPSTACKER_STATUS_PHASE_CALCULE_UPSTREAM_START_POSITION		:= 260,
	CSP_TRANSFER_UPSTACKER_STATUS_PHASE_MOVE_UPSTREAM_START_POSITION		:= 270,
	CSP_TRANSFER_UPSTACKER_STATUS_PHASE_MOVED_UPSTREAM_START_POSITION		:= 280,
	CSP_TRANSFER_UPSTACKER_STATUS_PHASE_CALCULE_DOWNSTREAM_START_POSITION_2	:= 281,
	CSP_TRANSFER_UPSTACKER_STATUS_PHASE_MOVE_DOWNSTREAM_START_POSITION_2	:= 282,
	CSP_TRANSFER_UPSTACKER_STATUS_PHASE_MOVED_DOWNSTREAM_START_POSITION_2	:= 283,
	CSP_TRANSFER_UPSTACKER_STATUS_PHASE_REDEFINE_MASTER_POSITION_STEP2		:= 290,
	CSP_TRANSFER_UPSTACKER_STATUS_PHASE_ENGAGE_DOWNSTREAM_STEP2				:= 300,
	CSP_TRANSFER_UPSTACKER_STATUS_PHASE_ENGAGE_UPSTREAM_STEP2				:= 310,
	CSP_TRANSFER_UPSTACKER_STATUS_PHASE_MOVE_MASTER_STEP2					:= 320,
	CSP_TRANSFER_UPSTACKER_STATUS_PHASE_DISENGAGE_STEP2						:= 330,
	CSP_TRANSFER_UPSTACKER_STATUS_PHASE_REDEFINE_MASTER_POSITION			:= 340,
	CSP_TRANSFER_UPSTACKER_STATUS_PHASE_MASTER_POSITION_REDEFINED			:= 350,
	CSP_TRANSFER_UPSTACKER_STATUS_PHASE_MOVE_PHASING						:= 400,
	CSP_TRANSFER_UPSTACKER_STATUS_PHASE_MOVED_PHASING						:= 410,	
	CSP_TRANSFER_UPSTACKER_STATUS_PHASE_CALCULATE_UPSTACKER_MASTER_POS		:= 415,	
	CSP_TRANSFER_UPSTACKER_STATUS_PHASE_CALCULATED_UPSTACKER_MASTER_POS_DONE:= 416,
	CSP_TRANSFER_UPSTACKER_STATUS_PHASE_REDFINE_MASTER_ABS_PHASE			:= 420,
	CSP_TRANSFER_UPSTACKER_STATUS_PHASE_ENGAGE_DOWNSTREAM					:= 500,
	CSP_TRANSFER_UPSTACKER_STATUS_PHASE_ENGAGE_UPSTREAM						:= 510,
	CSP_TRANSFER_UPSTACKER_STATUS_PHASE_MOVE_FINGER_LS						:= 512,
	CSP_TRANSFER_UPSTACKER_STATUS_PHASE_MOVE_FINGER_OS						:= 514,
	CSP_TRANSFER_UPSTACKER_STATUS_PHASE_ENGAGE_FINGER_LS					:= 520,
	CSP_TRANSFER_UPSTACKER_STATUS_PHASE_ENGAGE_FINGER_OS					:= 530,
	CSP_TRANSFER_UPSTACKER_STATUS_PHASE_ALL_ENGAGED							:= 540,
	CSP_TRANSFER_UPSTACKER_STATUS_PHASE_MOVE_MASTER_TO_IDLE					:= 550,
	CSP_TRANSFER_UPSTACKER_STATUS_PHASE_MOVED_MASTER_TO_IDLE				:= 560,
	CSP_TRANSFER_UPSTACKER_STATUS_PHASE_DONE 								:= 900,
	CSP_TRANSFER_UPSTACKER_STATUS_PHASE_ERROR 								:= 999
) := CSP_TRANSFER_UPSTACKER_STATUS_PHASE_START;
END_TYPE

// ---- Application/CSP/Transfer/Upstacker/csp_transfer_upstacker_status_enum.TcDUT
TYPE csp_transfer_upstacker_status_enum :
(
	CSP_TRANSFER_UPSTACKER_STATUS_NOT_INITIALIZED 							:=  0,
	CSP_TRANSFER_UPSTACKER_STATUS_DISABLED 									:=  10,
	CSP_TRANSFER_UPSTACKER_STATUS_ENABLE_REQUEST 							:=  20,
	CSP_TRANSFER_UPSTACKER_STATUS_ENABLING 									:=  30,
	CSP_TRANSFER_UPSTACKER_STATUS_ENABLED 									:=  40,
	CSP_TRANSFER_UPSTACKER_STATUS_HOME_REQUEST								:=  50,
	CSP_TRANSFER_UPSTACKER_STATUS_HOMING									:=  60,
	CSP_TRANSFER_UPSTACKER_STATUS_HOME_DONE									:=  70,
	CSP_TRANSFER_UPSTACKER_STATUS_CALCULATING_SLAVE_POSITION				:=  90,
	CSP_TRANSFER_UPSTACKER_STATUS_WAITING_SLAVE_ENGAGE						:= 100,
	CSP_TRANSFER_UPSTACKER_STATUS_PHASE_REQUEST								:= 140,
	CSP_TRANSFER_UPSTACKER_STATUS_PHASING									:= 150,
	CSP_TRANSFER_UPSTACKER_STATUS_PHASED									:= 160,
	CSP_TRANSFER_UPSTACKER_STATUS_CAM_ENGAGED_REQ							:= 170,
	CSP_TRANSFER_UPSTACKER_STATUS_AXIS_ENGAGE_VERIFY						:= 180,
	CSP_TRANSFER_UPSTACKER_STATUS_CAM_ON									:= 190,
	CSP_TRANSFER_UPSTACKER_STATUS_CAM_TABLE_READ							:= 195,
	CSP_TRANSFER_UPSTACKER_STATUS_CALCULATE_SLAVE_POSITION_REQUEST			:= 196,
	CSP_TRANSFER_UPSTACKER_STATUS_READY										:= 197,
	CSP_TRANSFER_UPSTACKER_STATUS_RUNNING_CAM								:= 200,
	CSP_TRANSFER_UPSTACKER_STATUS_CAM_OFF									:= 201,
	CSP_TRANSFER_UPSTACKER_STATUS_MOVING									:= 205,
	CSP_TRANSFER_UPSTACKER_STATUS_DISENGAGE									:= 210,
	CSP_TRANSFER_UPSTACKER_STATUS_DISENGAGING								:= 211,	
	CSP_TRANSFER_UPSTACKER_STATUS_STOP_REQUEST 								:= 500,
	CSP_TRANSFER_UPSTACKER_STATUS_DISABLE_REQUEST 							:= 530,
	CSP_TRANSFER_UPSTACKER_STATUS_DISABLING 								:= 540
) := CSP_TRANSFER_UPSTACKER_STATUS_NOT_INITIALIZED;
END_TYPE

// ---- Application/CSP/Transfer/Upstacker/csp_transfer_upstacker_test_status_enum.TcDUT
TYPE csp_transfer_upstacker_test_status_enum :
(		
	CSP_TRANSFER_UPSTACKER_STATUS_TEST_START								:= 0,
	CSP_TRANSFER_UPSTACKER_STATUS_TEST_DISABLE 								:= 10,
	CSP_TRANSFER_UPSTACKER_STATUS_TEST_ENABLE 								:= 20,
	CSP_TRANSFER_UPSTACKER_STATUS_TEST_ENABLED								:= 30,
	CSP_TRANSFER_UPSTACKER_STATUS_TEST_JOG_DOWNSTREAM						:= 40,
	CSP_TRANSFER_UPSTACKER_STATUS_TEST_REDEFINE_DOWNSTREAM					:= 50,
	CSP_TRANSFER_UPSTACKER_STATUS_TEST_JOG_UPSTREAM							:= 60,
	CSP_TRANSFER_UPSTACKER_STATUS_TEST_REDEFINE_UPSTREAM					:= 70,
	CSP_TRANSFER_UPSTACKER_STATUS_TEST_STOP 								:= 80,
	CSP_TRANSFER_UPSTACKER_STATUS_TEST_ERROR 								:= 999
) := CSP_TRANSFER_UPSTACKER_STATUS_TEST_START;
END_TYPE

// ---- Application/reject_reasons_enum.TcDUT
TYPE reject_reasons_enum :
(
	NO_REJ_REASON,	// 0 (this value must be the first of the list)
	POWER_UP_REJECT, // 1
	OPEN_FLAP_OPERATOR_SIDE, // 2
	OPEN_FLAP_LOADER_SIDE, // 3
	QUALITY_REJECT, // 4
	TRANSFER_CARTONS_HIGH_LOAD, //5
	OPEN_FLAP_OPERATOR_SIDE_INCHOERENCE, //6
	OPEN_FLAP_LOADER_SIDE_INCHOERENCE, //7
	TRAILING_MINOR_FLAP_OPEN, //8
	LEADING_MINOR_FLAP_OPEN, //9
	INCOMPLETE_GLUE //10
);
END_TYPE

// ---- Application/_Tasks/Application Status Manager/application_status_enum.TcDUT
TYPE application_status_enum : (
	APPLICATION_STATUS_NOT_INITIALIZED 					:= 0,	(*$ Initialization at power up to execute $*)
	APPLICATION_STATUS_1ST_POWERUP_ABSOLUTE				:= 1,
	APPLICATION_STATUS_1ST_POWERUP 						:= 2,
	APPLICATION_STATUS_2ND_POWERUP 						:= 3,
	APPLICATION_STATUS_3RD_POWERUP 						:= 4,
	APPLICATION_STATUS_RUNNING 							:= 5
	) := APPLICATION_STATUS_NOT_INITIALIZED;
END_TYPE

// ---- Data types/AFL extensions/analog_actuator/analog_actuator.TcDUT
(*   Copyright (c) 2007-2008 G.D SpA
*****************************************************************************************

Date:      Time:     | Author:   				|    Time spent: | Tester:   	   |  Time spent
*****************************************************************************************
*)
(*$
	The <i>analog_actuator</i> class abstracts a digital actuation with an optional digital feedback.<br/>
	The object is constructed with the <a href="#analog_actuator_init"><i>analog_actuator_init()</i></a> 
	method and feedbacks <a href="#digital_input_object"><i>digital_input</i></a> are optionally <br/>
	added through the two methods <a href="#analog_actuator_add_di_ready"><i>analog_actuator_add_di_ready()</i></a>
	and <a href="#analog_actuator_add_di_inactive"><i>analog_actuator_add_di_inactive()</i></a>.
	
	<p>
	If the active feedback is omitted then the actuator is declared active 
	(i.e. <a href="#analog_actuator_is_active"><i>analog_actuator_is_active()</i></a> = <i>TRUE</i>) <br/>
	after <a href="#analog_actuator_parameters"><i>active_time</i></a> parameter milliseconds are elapsed. <br/>
	The same happens with the <a href="#analog_actuator_parameters"><i>inactive_time</i></a> parameter if the 
	inactive feedback is omitted.
	</p>

	<p>
	It is important to understand the actuation model of the class that manages a one 
	<a href="#digital_output_object"><i>digital_output</i></a> object, <br/>
	so the only stable states are two: 
	<a href="#analog_actuator_status_enum"><i>ANALOG_ACTUATOR_STATUS_ACTIVE</i></a> and
	<a href="#analog_actuator_status_enum"><i>ANALOG_ACTUATOR_STATUS_INACTIVE</i></a>.
	</p>

</p>
	<p>
	See also: <br/>
	 <a href="#double_actuator_object"><i>double_actuator</i></a>
	</p>
$*)
(* Last used errorID_1 := 19 *)
TYPE
	analog_actuator:	STRUCT
	class_name:				STRING(MAX_OBJ_NAME_LENGTH) := ANALOG_ACTUATOR_CLASS_NAME;

	object_name:			STRING(MAX_OBJ_NAME_LENGTH) := '';

	descriptor:				descriptor;

	status:					analog_actuator_status_enum := ANALOG_ACTUATOR_STATUS_INIT;
	(*$M
	desc := Internal status of the analog_actuator: value among those defined in the <br/>
	enumerative <a href="#analog_actuator_status_enum"><i>analog_actuator_status_enum</i></a>; 
	$*)
	command:				analog_actuator_command_enum := ANALOG_ACTUATOR_CMD_INIT;
												(*$ Command that the analog_actuator
													is going to execute; value among
													those defined in the enumerative
													analog_actuator_command_enum $*)
	operational_command:	analog_actuator_command_enum := ANALOG_ACTUATOR_CMD_INIT;
												(*$ Command assigned when the analog_actuator
													is in the "operational" mode; value among
													those defined in the enumerative
													analog_actuator_command_enum $*)

	analog_physical_command: REAL := 0.0;

	test:					analog_actuator_test;
												(*$ This struct contains all the test's informations $*)

	di_ready:				POINTER TO digital_input;
	(*$U
	desc := Reference to the <a href="#digital_input_object"><i>digital_input</i></a>
	which check ready state (no alarm) of the analog_actuator.; 
	$*)

	ready_dchk:				digital_check;
	(*$I
	desc := if object has_di_ready is true, digital check is activated; 
	$*)

	di_active:				POINTER TO digital_input;
	(*$U
	desc := Reference to the <a href="#digital_input_object"><i>digital_input</i></a>
	which check active signal from the analog_actuator when do_activate is true.; 
	$*)

	active_dchk:			digital_check;
	(*$I
	desc := if object has_di_active is true and actuator is activated, digital check is activated; 
	$*)

	inactive_dchk:			digital_check;
	(*$I
	desc := if object has_di_active is true and actuator is inactive, digital check is activated; 
	$*)

	do_activate:			POINTER TO digital_output;
	(*$U
	desc := Reference to the <a href="#digital_output_object"><i>digital_output</i></a>
	which activates the analog_actuator.; 
	$*)

	ao_setpoint:			POINTER TO analog_output;
	(*$U
	desc := Reference to the <a href="#analog_output_object"><i>analog_output</i></a>
	which controls the analog output to the analog_actuator.; 
	$*)

	ai_feedback:			POINTER TO analog_input;
	(*$U
	desc := Reference to the <a href="#analog_input_object"><i>analog_input</i></a>
	which reads the feedback of the analog_actuator.; 
	$*)

	feedback_achk:			analog_check;
	(*$I
	desc := if object has_di_feedback is true, analog check is activated; 
	$*)

	feedback_upper_tolerance:	REAL := 10;		(*$P min :=  0; max :=  APPL; step := 1; unit := APPL;
													desc := Tolerance for upper feedback pyhsical value analog check. If the related feedback
													input is absent then this value is not used; 
												$*)

	feedback_lower_tolerance:	REAL := 10;		(*$P min :=  0; max :=  APPL; step := 1; unit := APPL;
													desc := Tolerance for lower feedback pyhsical value analog check. If the related feedback
													input is absent then this value is not used; 
												$*)

	has_di_ready:			BOOL := FALSE;		(*$ Info that states if the analog_actuator
													has the reference to a digital_input that
													performs ready status check; $*)

	has_di_active:			BOOL := FALSE;		(*$ Info that states if the analog_actuator
													has the reference to a digital_input that
													performs active status check; $*)

	has_do_activate:		BOOL := FALSE;		(*$ Info that states if the analog_actuator
													has the reference to the digital_output that
													performs the 'activation';
													must be	TRUE $*)

	has_ai_feedback:		BOOL := FALSE;		(*$ Info that states if the analog_actuator
													has the reference to a analog_input that
													performs feedback of the actuator; $*)

	is_active:				BOOL := FALSE;		(*$ Info that states the analog_actuator is active $*)
	is_inactive:			BOOL := FALSE;		(*$ Info that states the analog_actuator is inactive $*)
	timer:					timer;				(*$I desc :=  Timer to monitor activation/deactivation timeouts. ; $*)

	fault_reaction:			analog_actuator_fault_reaction_enum := ANALOG_ACTUATOR_FAULT_REACTION_DEACTIVATING;
												(*$ Fault reaction strategy. See 
													<a href="#analog_actuator_fault_reaction_enum"><i>reaction_enum</i></a> $*)
	active_time:			UDINT := 100;		(*$P min :=  0; max :=  APPL; step := 1; unit := ms;
													desc := Activation timeout. If the related feedback
													input is absent then this value is used to declare
													<a href="#analog_actuator_status_enum"><i>INACTIVE</i></a>; 
												$*)

	inactive_time:			UDINT := 100;		(*$P min :=  0; max :=  APPL; step := 1; unit := ms;
													desc := Deactivation timeout. If the related feedback
													input is absent then this value is used to declare
													<a href="#analog_actuator_status_enum"><i>INACTIVE</i></a>; 
											    $*)
	out_of_lower_range_fem:	analog_actuator_snapshot;

